// SIMATIC STEP 7 (V5.x) project PLC_KIP
// CPU: CPU 317-2 PN/DP
// station: Hardware
// station: VIPA
// station: P_ADR_BUS
// program: S7 Program(1)

SYMBOL_TABLE
"empty_C0"	C 0	COUNTER
"dFilt_cnt"	C 1	COUNTER
"COM"	DB 100	DB 100
"znm15_pid"	DB 500	FB 58
"CV_dConc1_pid"	DB 501	FB 58
"zadv_riv_nya"	DB 502	FB 58
"Dat_Filt"	FB 1	FB 1
"MD_to_MW"	FB 2	FB 2
"DO_Control"	FB 3	FB 3
"DI_DO_STATE"	FB 4	FB 4
"PID_AO_control"	FB 5	FB 5
"dat_alm"	FB 6	FB 6
"PUT"	FB 15	FB 15	// Write Data to a Remote CPU
"TCONT_CP"	FB 58	FB 58	// temperature PID controller with pulse generator and self-tuning
"DO_MANUAL"	FC 1	FC 1
"SCALE"	FC 105	FC 105	// Scaling Values
"UNSCALE"	FC 106	FC 106	// Unscaling Values
"btn_kvit"	M 3998.0	BOOL
"ZNM15_HM"	M 6000.1	BOOL
"CYCL_EXC"	OB 1	OB 1	// Cycle Execution
"CYC_INT5"	OB 35	OB 35	// Cyclic Interrupt 5
"AIt1_1"	PIW 272	INT
"AIt1_2"	PIW 274	INT
"AIt1_3"	PIW 276	INT
"AIt1_4"	PIW 278	INT
"AIt2_1"	PIW 280	INT
"AIt2_2"	PIW 282	INT
"AIt2_3"	PIW 284	INT
"AIt2_4"	PIW 286	INT
"AIt_3_1"	PIW 288	INT
"AIt_3_2"	PIW 290	INT
"AIt3_3"	PIW 292	INT
"AIt3_4"	PIW 294	INT
"ZN1_cur"	PIW 304	INT
"UVK2_cur"	PIW 306	INT
"UVK1_cur"	PIW 308	INT
"UZ1_in"	PIW 310	INT
"UZ1_out"	PIW 312	INT
"vak_suk1"	PIW 314	INT
"Pidsit_riv"	PIW 316	INT
"vak_suk2"	PIW 318	INT
"vak_suk3"	PIW 320	INT
"vak_suk5"	PIW 322	INT
"vak_suk4"	PIW 324	INT
"vak_suk6"	PIW 326	INT
"vak_val1"	PIW 328	INT
"vak_VN5"	PIW 330	INT
"vak_val2"	PIW 332	INT
"BM8_riv"	PIW 334	INT
"BO9_riv"	PIW 336	INT
"BB11_riv"	PIW 338	INT
"BZ10_riv"	PIW 340	INT
"Gauch_riv"	PIW 342	INT
"NC32"	PIW 344	INT
"Priam_riv"	PIW 346	INT
"NC35"	PIW 348	INT
"GRG_riv"	PIW 350	INT
"vak_VN1"	PIW 352	INT
"vak_VN3"	PIW 354	INT
"vak_VN2"	PIW 356	INT
"vak_VN4"	PIW 358	INT
"dUVK1_in"	PIW 376	INT
"dUVK2_in"	PIW 378	INT
"dC8_in"	PIW 380	INT
"dUVK1_out"	PIW 382	INT
"dUVK2_out"	PIW 384	INT
"dC8_out"	PIW 386	INT
"dSUM_pr"	PIW 388	INT
"AI2_4"	PIW 390	INT
"dRivSkop"	PIW 392	INT
"dRIV_NYA"	PIW 394	INT
"dRivPidNya"	PIW 396	INT
"dUzloulov_in"	PIW 398	INT
"dMlyn_in"	PIW 400	INT
"AI4_2"	PIW 402	INT
"dMlyn_out"	PIW 404	INT
"dUzloulov_out"	PIW 406	INT
"taskZNM12"	PQW 272	INT
"ZasNV23_1"	PQW 274	INT
"taskZNM15"	PQW 276	INT
"reg_knctr2"	PQW 278	INT
"zadv_recycl_nya"	PQW 296	INT
"CV_conc1"	PQW 300	INT
"GET"	SFB 14	SFB 14	// Read Data From a Remote CPU
"empty_T0"	T 0	TIMER
"dFilt_tmr"	T 1	TIMER
"VAT_3_kip"	VAT 1	
"VAT_4"	VAT 2	
"VAT_3_HI_LOW_Dat"	VAT 3	
END_SYMBOL_TABLE

FUNCTION_BLOCK "Dat_Filt"	// FB 1
TITLE = Чтение датчика
//**********************************
VERSION : 0.1
VAR_INPUT
  dPIW : INT ;
  dHi_lim : DINT ;
  dLow_lim : DINT ;
  dErr_lvl : INT ;
  Sample : S5TIME ;
END_VAR
VAR_OUTPUT
  Dat_err : BOOL ;
  Dat_f : REAL ;
  Dat_md : DINT ;
END_VAR
VAR
  Bipolar : BOOL ;
  rst_T1 : BOOL ;
  int_C1 : INT ;
  Hi_lim_re : REAL ;
  Low_lim_re : REAL ;
  DAT_re : REAL ;
  DAT_avg : REAL ;
  dat_re0 : REAL ;
  dat_re1 : REAL ;
  dat_re2 : REAL ;
  dat_re3 : REAL ;
  dat_re4 : REAL ;
  dat_re5 : REAL ;
  dat_re6 : REAL ;
  dat_re7 : REAL ;
  dat_re8 : REAL ;
  dat_re9 : REAL ;
  sum : REAL ;
END_VAR
VAR_TEMP
  SCL_err : WORD ;
  UNSCL_err : WORD ;
END_VAR
BEGIN
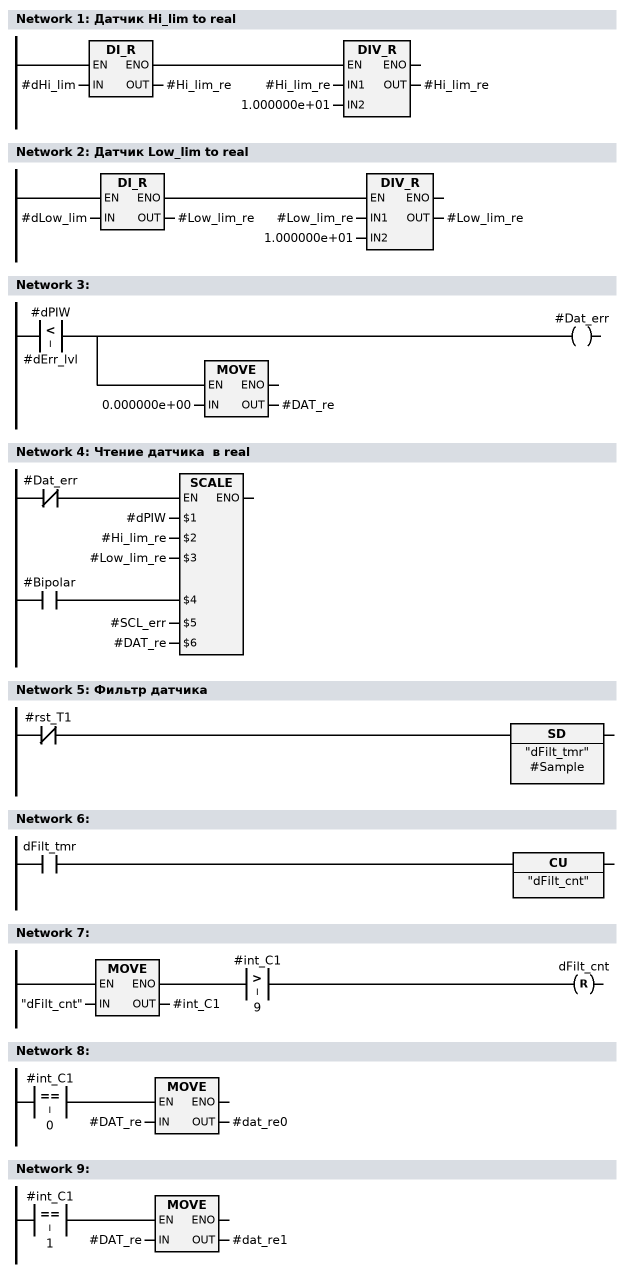
NETWORK
TITLE = Датчик Hi_lim to real
      A(;
      L     #dHi_lim;
      DTR;
      T     #Hi_lim_re;
      SET;
      SAVE;
      CLR;
      A     BR;
      );
      JNB   _001;
      L     #Hi_lim_re;
      L     1.000000e+01;
      /R;
      T     #Hi_lim_re;
_001: NOP   0;
NETWORK
TITLE = Датчик Low_lim to real
      A(;
      L     #dLow_lim;
      DTR;
      T     #Low_lim_re;
      SET;
      SAVE;
      CLR;
      A     BR;
      );
      JNB   _002;
      L     #Low_lim_re;
      L     1.000000e+01;
      /R;
      T     #Low_lim_re;
_002: NOP   0;
NETWORK
TITLE =
//Ошибка чтения датчика
      L     #dPIW;
      L     #dErr_lvl;
      <I;
      =     L 4.0;
      A     L 4.0;
      BLD   102;
      =     #Dat_err;
      A     L 4.0;
      JNB   _003;
      L     0.000000e+00;
      T     #DAT_re;
_003: NOP   0;
NETWORK
TITLE = Чтение датчика  в real
      A     #Bipolar;
      =     L 4.0;
      BLD   103;
      AN    #Dat_err;
      JNB   _004;
      CALL  "SCALE" (
           $1                       := #dPIW,
           $2                       := #Hi_lim_re,
           $3                       := #Low_lim_re,
           $4                       := L 4.0,
           $5                       := #SCL_err,
           $6                       := #DAT_re);
_004: NOP   0;
NETWORK
TITLE = Фильтр датчика
//***************************************************
      AN    #rst_T1;
      L     #Sample;
      SD    "dFilt_tmr";
NETWORK
TITLE =
      A     "dFilt_tmr";
      CU    "dFilt_cnt";
NETWORK
TITLE =
      A(;
      L     "dFilt_cnt";
      T     #int_C1;
      SET;
      SAVE;
      CLR;
      A     BR;
      );
      A(;
      L     #int_C1;
      L     9;
      >I;
      );
      R     "dFilt_cnt";
NETWORK
TITLE =
      A(;
      L     #int_C1;
      L     0;
      ==I;
      );
      JNB   _005;
      L     #DAT_re;
      T     #dat_re0;
_005: NOP   0;
NETWORK
TITLE =
      A(;
      L     #int_C1;
      L     1;
      ==I;
      );
      JNB   _006;
      L     #DAT_re;
      T     #dat_re1;
_006: NOP   0;
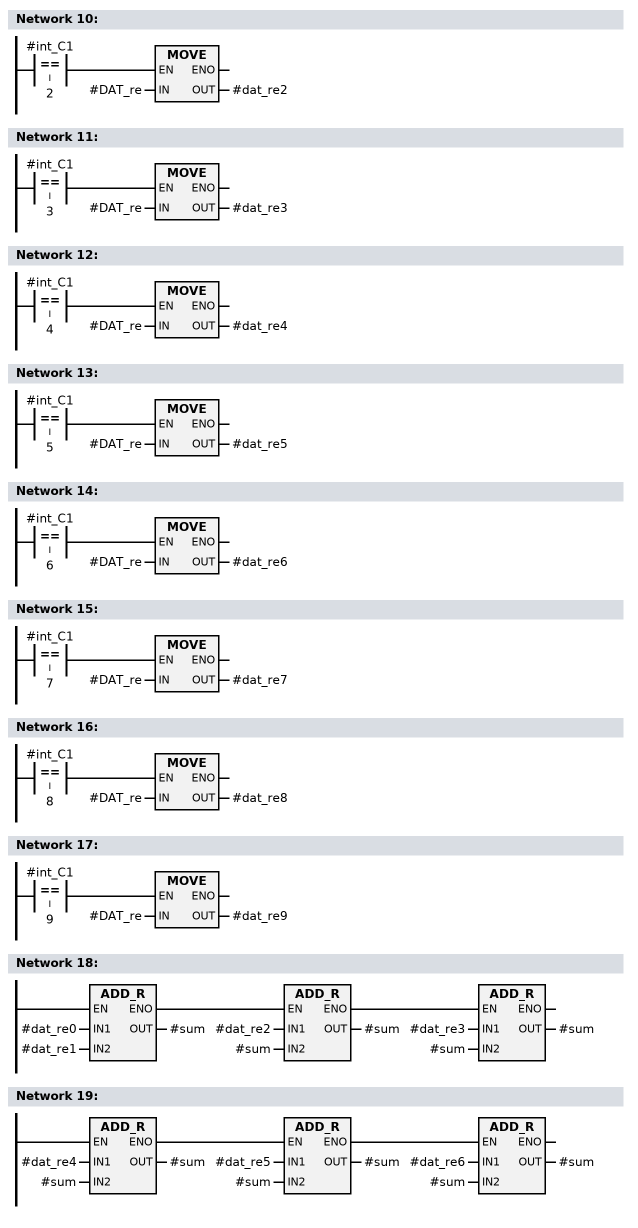
NETWORK
TITLE =
      A(;
      L     #int_C1;
      L     2;
      ==I;
      );
      JNB   _007;
      L     #DAT_re;
      T     #dat_re2;
_007: NOP   0;
NETWORK
TITLE =
      A(;
      L     #int_C1;
      L     3;
      ==I;
      );
      JNB   _008;
      L     #DAT_re;
      T     #dat_re3;
_008: NOP   0;
NETWORK
TITLE =
      A(;
      L     #int_C1;
      L     4;
      ==I;
      );
      JNB   _009;
      L     #DAT_re;
      T     #dat_re4;
_009: NOP   0;
NETWORK
TITLE =
      A(;
      L     #int_C1;
      L     5;
      ==I;
      );
      JNB   _00a;
      L     #DAT_re;
      T     #dat_re5;
_00a: NOP   0;
NETWORK
TITLE =
      A(;
      L     #int_C1;
      L     6;
      ==I;
      );
      JNB   _00b;
      L     #DAT_re;
      T     #dat_re6;
_00b: NOP   0;
NETWORK
TITLE =
      A(;
      L     #int_C1;
      L     7;
      ==I;
      );
      JNB   _00c;
      L     #DAT_re;
      T     #dat_re7;
_00c: NOP   0;
NETWORK
TITLE =
      A(;
      L     #int_C1;
      L     8;
      ==I;
      );
      JNB   _00d;
      L     #DAT_re;
      T     #dat_re8;
_00d: NOP   0;
NETWORK
TITLE =
      A(;
      L     #int_C1;
      L     9;
      ==I;
      );
      JNB   _00e;
      L     #DAT_re;
      T     #dat_re9;
_00e: NOP   0;
NETWORK
TITLE =
      A(;
      A(;
      L     #dat_re0;
      L     #dat_re1;
      +R;
      T     #sum;
      AN    OV;
      SAVE;
      CLR;
      A     BR;
      );
      JNB   _00f;
      L     #dat_re2;
      L     #sum;
      +R;
      T     #sum;
      AN    OV;
      SAVE;
      CLR;
_00f: A     BR;
      );
      JNB   _010;
      L     #dat_re3;
      L     #sum;
      +R;
      T     #sum;
_010: NOP   0;
NETWORK
TITLE =
      A(;
      A(;
      L     #dat_re4;
      L     #sum;
      +R;
      T     #sum;
      AN    OV;
      SAVE;
      CLR;
      A     BR;
      );
      JNB   _011;
      L     #dat_re5;
      L     #sum;
      +R;
      T     #sum;
      AN    OV;
      SAVE;
      CLR;
_011: A     BR;
      );
      JNB   _012;
      L     #dat_re6;
      L     #sum;
      +R;
      T     #sum;
_012: NOP   0;
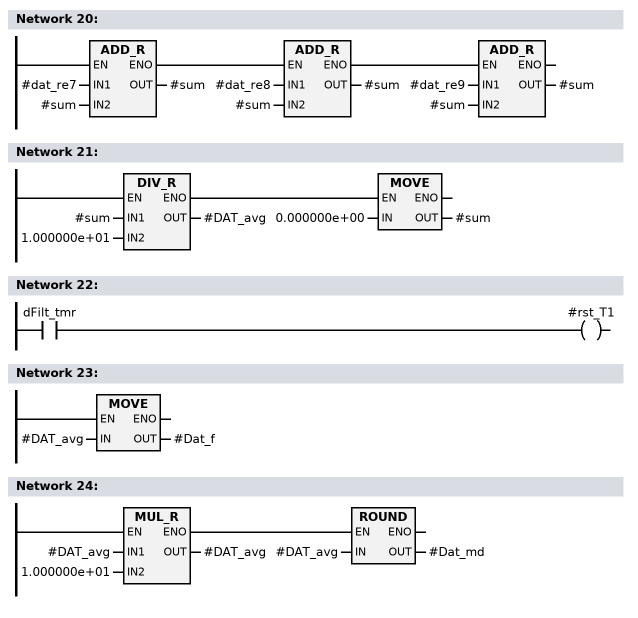
NETWORK
TITLE =
      A(;
      A(;
      L     #dat_re7;
      L     #sum;
      +R;
      T     #sum;
      AN    OV;
      SAVE;
      CLR;
      A     BR;
      );
      JNB   _013;
      L     #dat_re8;
      L     #sum;
      +R;
      T     #sum;
      AN    OV;
      SAVE;
      CLR;
_013: A     BR;
      );
      JNB   _014;
      L     #dat_re9;
      L     #sum;
      +R;
      T     #sum;
_014: NOP   0;
NETWORK
TITLE =
      A(;
      L     #sum;
      L     1.000000e+01;
      /R;
      T     #DAT_avg;
      AN    OV;
      SAVE;
      CLR;
      A     BR;
      );
      JNB   _015;
      L     0.000000e+00;
      T     #sum;
_015: NOP   0;
NETWORK
TITLE =
      A     "dFilt_tmr";
      =     #rst_T1;
NETWORK
TITLE =
      L     #DAT_avg;
      T     #Dat_f;
      NOP   0;
NETWORK
TITLE =
      A(;
      L     #DAT_avg;
      L     1.000000e+01;
      *R;
      T     #DAT_avg;
      AN    OV;
      SAVE;
      CLR;
      A     BR;
      );
      JNB   _016;
      L     #DAT_avg;
      RND;
      T     #Dat_md;
_016: NOP   0;
END_FUNCTION_BLOCK

FUNCTION_BLOCK "MD_to_MW"	// FB 2
//Для обміну між ПЛК КІП та ПЛК ДВГ (з MD в MW)
VERSION : 0.1
VAR_TEMP
  ZNM15_task_re : REAL ;
  cv_conc1_task_re : REAL ;
  cv_recycle_task_re : REAL ;
END_VAR
BEGIN
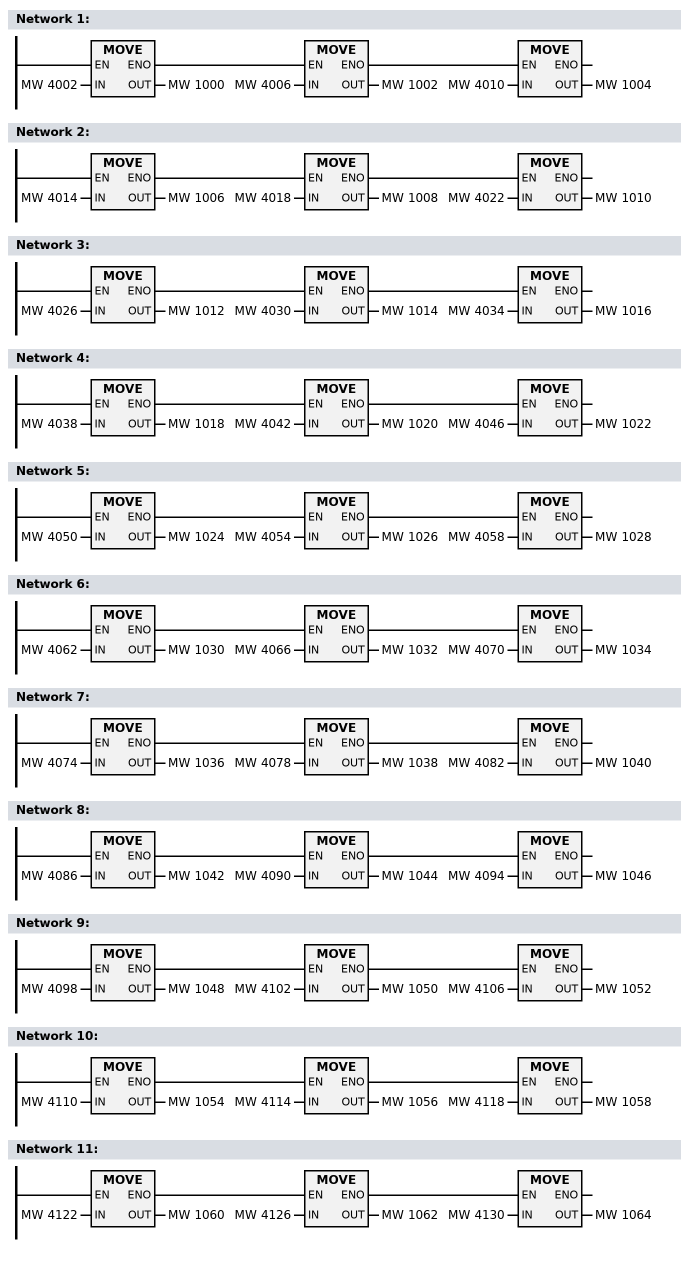
NETWORK
TITLE =
      A(;
      A(;
      L     MW 4002;
      T     MW 1000;
      SET;
      SAVE;
      CLR;
      A     BR;
      );
      JNB   _001;
      L     MW 4006;
      T     MW 1002;
      SET;
      SAVE;
      CLR;
_001: A     BR;
      );
      JNB   _002;
      L     MW 4010;
      T     MW 1004;
_002: NOP   0;
NETWORK
TITLE =
      A(;
      A(;
      L     MW 4014;
      T     MW 1006;
      SET;
      SAVE;
      CLR;
      A     BR;
      );
      JNB   _003;
      L     MW 4018;
      T     MW 1008;
      SET;
      SAVE;
      CLR;
_003: A     BR;
      );
      JNB   _004;
      L     MW 4022;
      T     MW 1010;
_004: NOP   0;
NETWORK
TITLE =
      A(;
      A(;
      L     MW 4026;
      T     MW 1012;
      SET;
      SAVE;
      CLR;
      A     BR;
      );
      JNB   _005;
      L     MW 4030;
      T     MW 1014;
      SET;
      SAVE;
      CLR;
_005: A     BR;
      );
      JNB   _006;
      L     MW 4034;
      T     MW 1016;
_006: NOP   0;
NETWORK
TITLE =
      A(;
      A(;
      L     MW 4038;
      T     MW 1018;
      SET;
      SAVE;
      CLR;
      A     BR;
      );
      JNB   _007;
      L     MW 4042;
      T     MW 1020;
      SET;
      SAVE;
      CLR;
_007: A     BR;
      );
      JNB   _008;
      L     MW 4046;
      T     MW 1022;
_008: NOP   0;
NETWORK
TITLE =
      A(;
      A(;
      L     MW 4050;
      T     MW 1024;
      SET;
      SAVE;
      CLR;
      A     BR;
      );
      JNB   _009;
      L     MW 4054;
      T     MW 1026;
      SET;
      SAVE;
      CLR;
_009: A     BR;
      );
      JNB   _00a;
      L     MW 4058;
      T     MW 1028;
_00a: NOP   0;
NETWORK
TITLE =
      A(;
      A(;
      L     MW 4062;
      T     MW 1030;
      SET;
      SAVE;
      CLR;
      A     BR;
      );
      JNB   _00b;
      L     MW 4066;
      T     MW 1032;
      SET;
      SAVE;
      CLR;
_00b: A     BR;
      );
      JNB   _00c;
      L     MW 4070;
      T     MW 1034;
_00c: NOP   0;
NETWORK
TITLE =
      A(;
      A(;
      L     MW 4074;
      T     MW 1036;
      SET;
      SAVE;
      CLR;
      A     BR;
      );
      JNB   _00d;
      L     MW 4078;
      T     MW 1038;
      SET;
      SAVE;
      CLR;
_00d: A     BR;
      );
      JNB   _00e;
      L     MW 4082;
      T     MW 1040;
_00e: NOP   0;
NETWORK
TITLE =
      A(;
      A(;
      L     MW 4086;
      T     MW 1042;
      SET;
      SAVE;
      CLR;
      A     BR;
      );
      JNB   _00f;
      L     MW 4090;
      T     MW 1044;
      SET;
      SAVE;
      CLR;
_00f: A     BR;
      );
      JNB   _010;
      L     MW 4094;
      T     MW 1046;
_010: NOP   0;
NETWORK
TITLE =
      A(;
      A(;
      L     MW 4098;
      T     MW 1048;
      SET;
      SAVE;
      CLR;
      A     BR;
      );
      JNB   _011;
      L     MW 4102;
      T     MW 1050;
      SET;
      SAVE;
      CLR;
_011: A     BR;
      );
      JNB   _012;
      L     MW 4106;
      T     MW 1052;
_012: NOP   0;
NETWORK
TITLE =
      A(;
      A(;
      L     MW 4110;
      T     MW 1054;
      SET;
      SAVE;
      CLR;
      A     BR;
      );
      JNB   _013;
      L     MW 4114;
      T     MW 1056;
      SET;
      SAVE;
      CLR;
_013: A     BR;
      );
      JNB   _014;
      L     MW 4118;
      T     MW 1058;
_014: NOP   0;
NETWORK
TITLE =
      A(;
      A(;
      L     MW 4122;
      T     MW 1060;
      SET;
      SAVE;
      CLR;
      A     BR;
      );
      JNB   _015;
      L     MW 4126;
      T     MW 1062;
      SET;
      SAVE;
      CLR;
_015: A     BR;
      );
      JNB   _016;
      L     MW 4130;
      T     MW 1064;
_016: NOP   0;
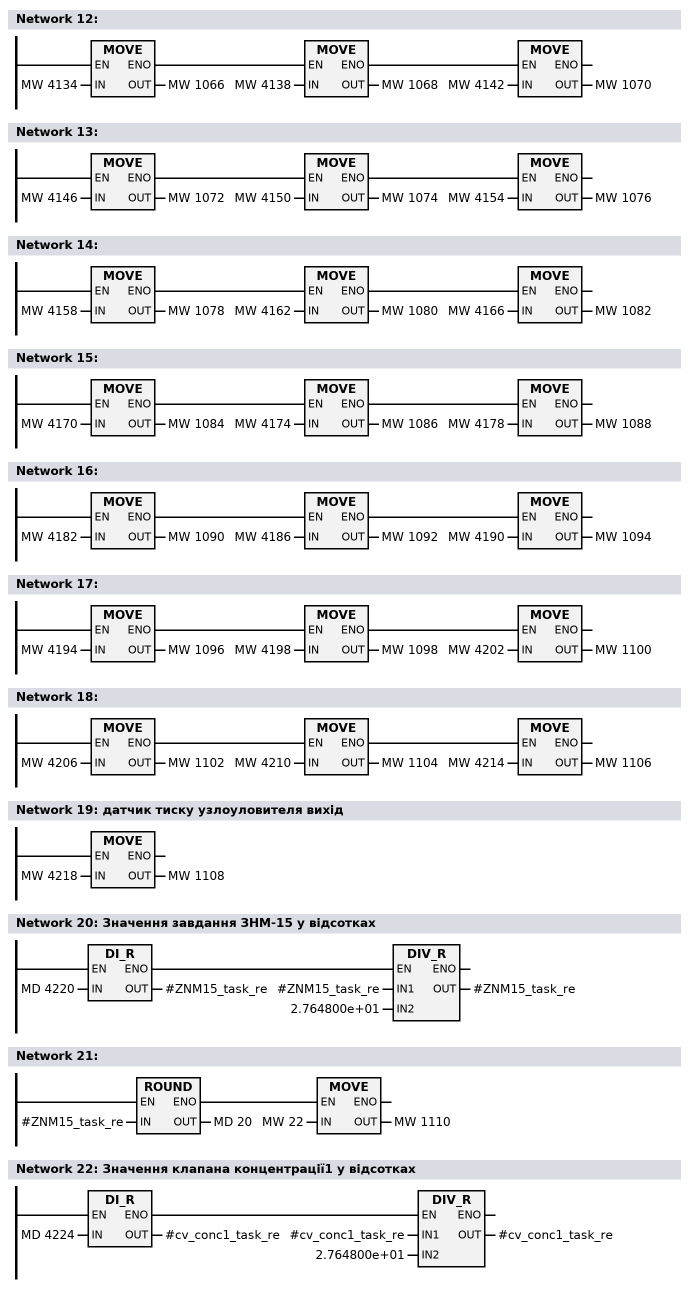
NETWORK
TITLE =
      A(;
      A(;
      L     MW 4134;
      T     MW 1066;
      SET;
      SAVE;
      CLR;
      A     BR;
      );
      JNB   _017;
      L     MW 4138;
      T     MW 1068;
      SET;
      SAVE;
      CLR;
_017: A     BR;
      );
      JNB   _018;
      L     MW 4142;
      T     MW 1070;
_018: NOP   0;
NETWORK
TITLE =
      A(;
      A(;
      L     MW 4146;
      T     MW 1072;
      SET;
      SAVE;
      CLR;
      A     BR;
      );
      JNB   _019;
      L     MW 4150;
      T     MW 1074;
      SET;
      SAVE;
      CLR;
_019: A     BR;
      );
      JNB   _01a;
      L     MW 4154;
      T     MW 1076;
_01a: NOP   0;
NETWORK
TITLE =
      A(;
      A(;
      L     MW 4158;
      T     MW 1078;
      SET;
      SAVE;
      CLR;
      A     BR;
      );
      JNB   _01b;
      L     MW 4162;
      T     MW 1080;
      SET;
      SAVE;
      CLR;
_01b: A     BR;
      );
      JNB   _01c;
      L     MW 4166;
      T     MW 1082;
_01c: NOP   0;
NETWORK
TITLE =
      A(;
      A(;
      L     MW 4170;
      T     MW 1084;
      SET;
      SAVE;
      CLR;
      A     BR;
      );
      JNB   _01d;
      L     MW 4174;
      T     MW 1086;
      SET;
      SAVE;
      CLR;
_01d: A     BR;
      );
      JNB   _01e;
      L     MW 4178;
      T     MW 1088;
_01e: NOP   0;
NETWORK
TITLE =
      A(;
      A(;
      L     MW 4182;
      T     MW 1090;
      SET;
      SAVE;
      CLR;
      A     BR;
      );
      JNB   _01f;
      L     MW 4186;
      T     MW 1092;
      SET;
      SAVE;
      CLR;
_01f: A     BR;
      );
      JNB   _020;
      L     MW 4190;
      T     MW 1094;
_020: NOP   0;
NETWORK
TITLE =
      A(;
      A(;
      L     MW 4194;
      T     MW 1096;
      SET;
      SAVE;
      CLR;
      A     BR;
      );
      JNB   _021;
      L     MW 4198;
      T     MW 1098;
      SET;
      SAVE;
      CLR;
_021: A     BR;
      );
      JNB   _022;
      L     MW 4202;
      T     MW 1100;
_022: NOP   0;
NETWORK
TITLE =
      A(;
      A(;
      L     MW 4206;
      T     MW 1102;
      SET;
      SAVE;
      CLR;
      A     BR;
      );
      JNB   _023;
      L     MW 4210;
      T     MW 1104;
      SET;
      SAVE;
      CLR;
_023: A     BR;
      );
      JNB   _024;
      L     MW 4214;
      T     MW 1106;
_024: NOP   0;
NETWORK
TITLE = датчик тиску узлоуловителя вихід
      L     MW 4218;
      T     MW 1108;
      NOP   0;
NETWORK
TITLE = Значення завдання ЗНМ-15 у відсотках
//Значення завдання ЗНМ-15 у відсотках
      A(;
      L     MD 4220;
      DTR;
      T     #ZNM15_task_re;
      SET;
      SAVE;
      CLR;
      A     BR;
      );
      JNB   _025;
      L     #ZNM15_task_re;
      L     2.764800e+01;
      /R;
      T     #ZNM15_task_re;
_025: NOP   0;
NETWORK
TITLE =
      A(;
      L     #ZNM15_task_re;
      RND;
      T     MD 20;
      AN    OV;
      SAVE;
      CLR;
      A     BR;
      );
      JNB   _026;
      L     MW 22;
      T     MW 1110;
_026: NOP   0;
NETWORK
TITLE = Значення клапана концентрації1 у відсотках
      A(;
      L     MD 4224;
      DTR;
      T     #cv_conc1_task_re;
      SET;
      SAVE;
      CLR;
      A     BR;
      );
      JNB   _027;
      L     #cv_conc1_task_re;
      L     2.764800e+01;
      /R;
      T     #cv_conc1_task_re;
_027: NOP   0;
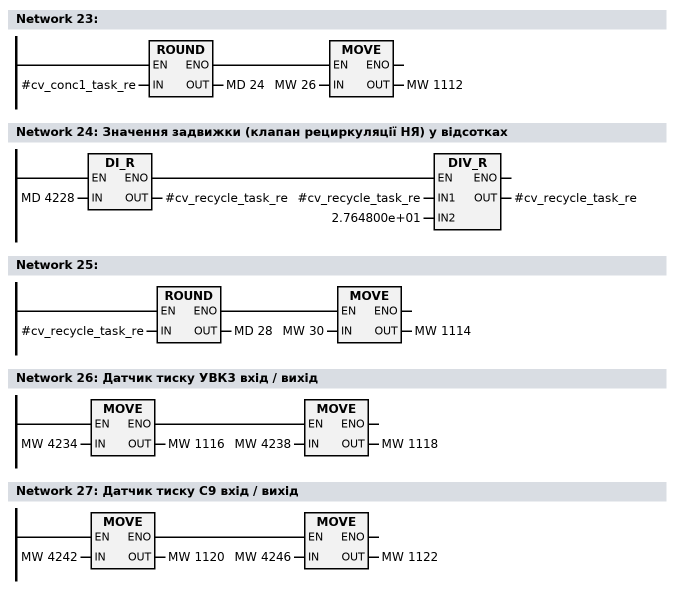
NETWORK
TITLE =
      A(;
      L     #cv_conc1_task_re;
      RND;
      T     MD 24;
      AN    OV;
      SAVE;
      CLR;
      A     BR;
      );
      JNB   _028;
      L     MW 26;
      T     MW 1112;
_028: NOP   0;
NETWORK
TITLE = Значення задвижки (клапан рециркуляції НЯ) у відсотках
      A(;
      L     MD 4228;
      DTR;
      T     #cv_recycle_task_re;
      SET;
      SAVE;
      CLR;
      A     BR;
      );
      JNB   _029;
      L     #cv_recycle_task_re;
      L     2.764800e+01;
      /R;
      T     #cv_recycle_task_re;
_029: NOP   0;
NETWORK
TITLE =
      A(;
      L     #cv_recycle_task_re;
      RND;
      T     MD 28;
      AN    OV;
      SAVE;
      CLR;
      A     BR;
      );
      JNB   _02a;
      L     MW 30;
      T     MW 1114;
_02a: NOP   0;
NETWORK
TITLE = Датчик тиску УВК3 вхід / вихід
      A(;
      L     MW 4234;
      T     MW 1116;
      SET;
      SAVE;
      CLR;
      A     BR;
      );
      JNB   _02b;
      L     MW 4238;
      T     MW 1118;
_02b: NOP   0;
NETWORK
TITLE = Датчик тиску C9 вхід / вихід
      A(;
      L     MW 4242;
      T     MW 1120;
      SET;
      SAVE;
      CLR;
      A     BR;
      );
      JNB   _02c;
      L     MW 4246;
      T     MW 1122;
_02c: NOP   0;
END_FUNCTION_BLOCK

FUNCTION_BLOCK "DO_Control"	// FB 3
//Керування дискретними виходами
VERSION : 0.1
BEGIN
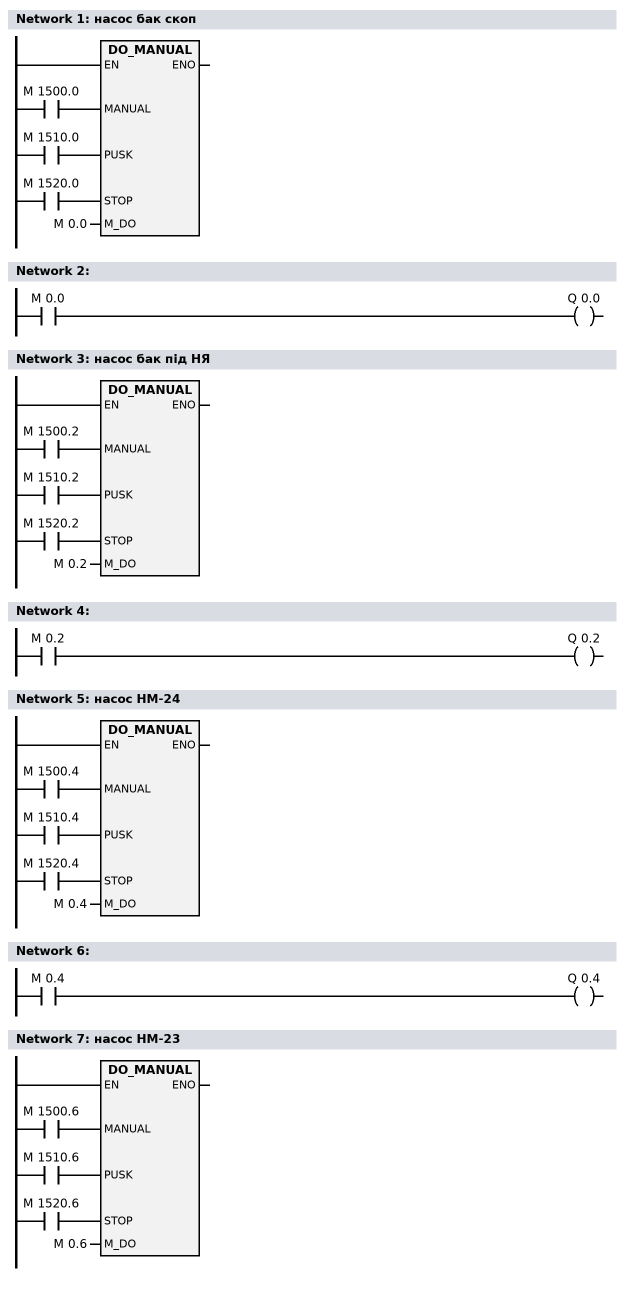
NETWORK
TITLE = насос бак скоп
      A     M 1500.0;
      =     L 0.0;
      BLD   103;
      A     M 1510.0;
      =     L 0.1;
      BLD   103;
      A     M 1520.0;
      =     L 0.2;
      BLD   103;
      CALL  "DO_MANUAL" (
           MANUAL                   := L 0.0,
           PUSK                     := L 0.1,
           STOP                     := L 0.2,
           M_DO                     := M 0.0);
      NOP   0;
NETWORK
TITLE =
      A     M 0.0;
      =     Q 0.0;
NETWORK
TITLE = насос бак під НЯ
      A     M 1500.2;
      =     L 0.0;
      BLD   103;
      A     M 1510.2;
      =     L 0.1;
      BLD   103;
      A     M 1520.2;
      =     L 0.2;
      BLD   103;
      CALL  "DO_MANUAL" (
           MANUAL                   := L 0.0,
           PUSK                     := L 0.1,
           STOP                     := L 0.2,
           M_DO                     := M 0.2);
      NOP   0;
NETWORK
TITLE =
      A     M 0.2;
      =     Q 0.2;
NETWORK
TITLE = насос НМ-24
      A     M 1500.4;
      =     L 0.0;
      BLD   103;
      A     M 1510.4;
      =     L 0.1;
      BLD   103;
      A     M 1520.4;
      =     L 0.2;
      BLD   103;
      CALL  "DO_MANUAL" (
           MANUAL                   := L 0.0,
           PUSK                     := L 0.1,
           STOP                     := L 0.2,
           M_DO                     := M 0.4);
      NOP   0;
NETWORK
TITLE =
      A     M 0.4;
      =     Q 0.4;
NETWORK
TITLE = насос НМ-23
      A     M 1500.6;
      =     L 0.0;
      BLD   103;
      A     M 1510.6;
      =     L 0.1;
      BLD   103;
      A     M 1520.6;
      =     L 0.2;
      BLD   103;
      CALL  "DO_MANUAL" (
           MANUAL                   := L 0.0,
           PUSK                     := L 0.1,
           STOP                     := L 0.2,
           M_DO                     := M 0.6);
      NOP   0;
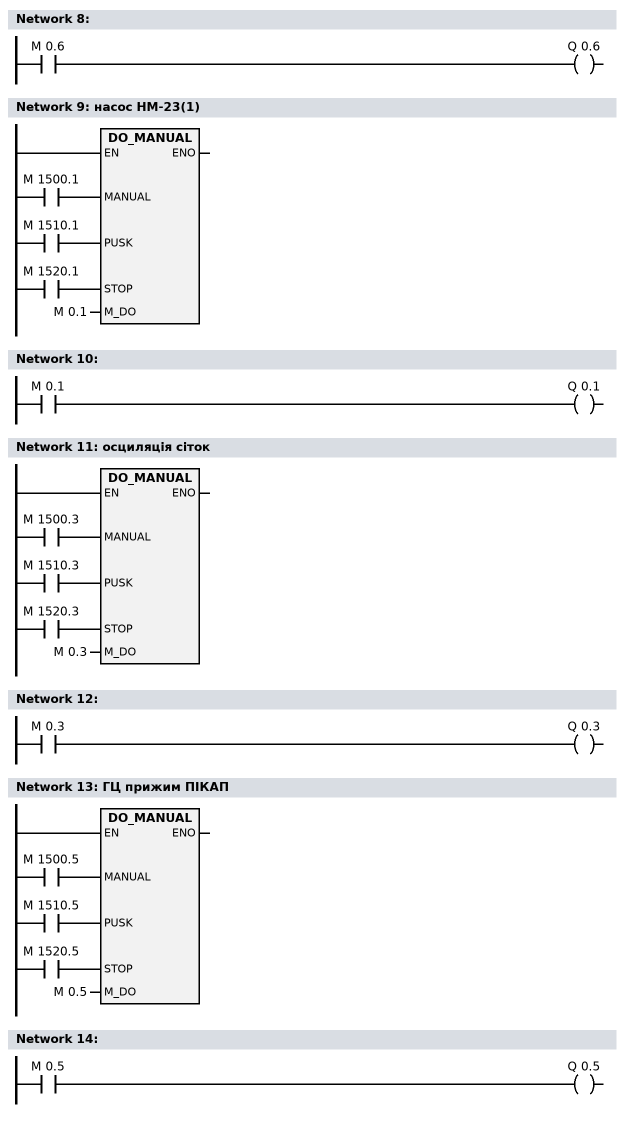
NETWORK
TITLE =
      A     M 0.6;
      =     Q 0.6;
NETWORK
TITLE = насос НМ-23(1)
      A     M 1500.1;
      =     L 0.0;
      BLD   103;
      A     M 1510.1;
      =     L 0.1;
      BLD   103;
      A     M 1520.1;
      =     L 0.2;
      BLD   103;
      CALL  "DO_MANUAL" (
           MANUAL                   := L 0.0,
           PUSK                     := L 0.1,
           STOP                     := L 0.2,
           M_DO                     := M 0.1);
      NOP   0;
NETWORK
TITLE =
      A     M 0.1;
      =     Q 0.1;
NETWORK
TITLE = осциляція сіток
      A     M 1500.3;
      =     L 0.0;
      BLD   103;
      A     M 1510.3;
      =     L 0.1;
      BLD   103;
      A     M 1520.3;
      =     L 0.2;
      BLD   103;
      CALL  "DO_MANUAL" (
           MANUAL                   := L 0.0,
           PUSK                     := L 0.1,
           STOP                     := L 0.2,
           M_DO                     := M 0.3);
      NOP   0;
NETWORK
TITLE =
      A     M 0.3;
      =     Q 0.3;
NETWORK
TITLE = ГЦ прижим ПІКАП
      A     M 1500.5;
      =     L 0.0;
      BLD   103;
      A     M 1510.5;
      =     L 0.1;
      BLD   103;
      A     M 1520.5;
      =     L 0.2;
      BLD   103;
      CALL  "DO_MANUAL" (
           MANUAL                   := L 0.0,
           PUSK                     := L 0.1,
           STOP                     := L 0.2,
           M_DO                     := M 0.5);
      NOP   0;
NETWORK
TITLE =
      A     M 0.5;
      =     Q 0.5;
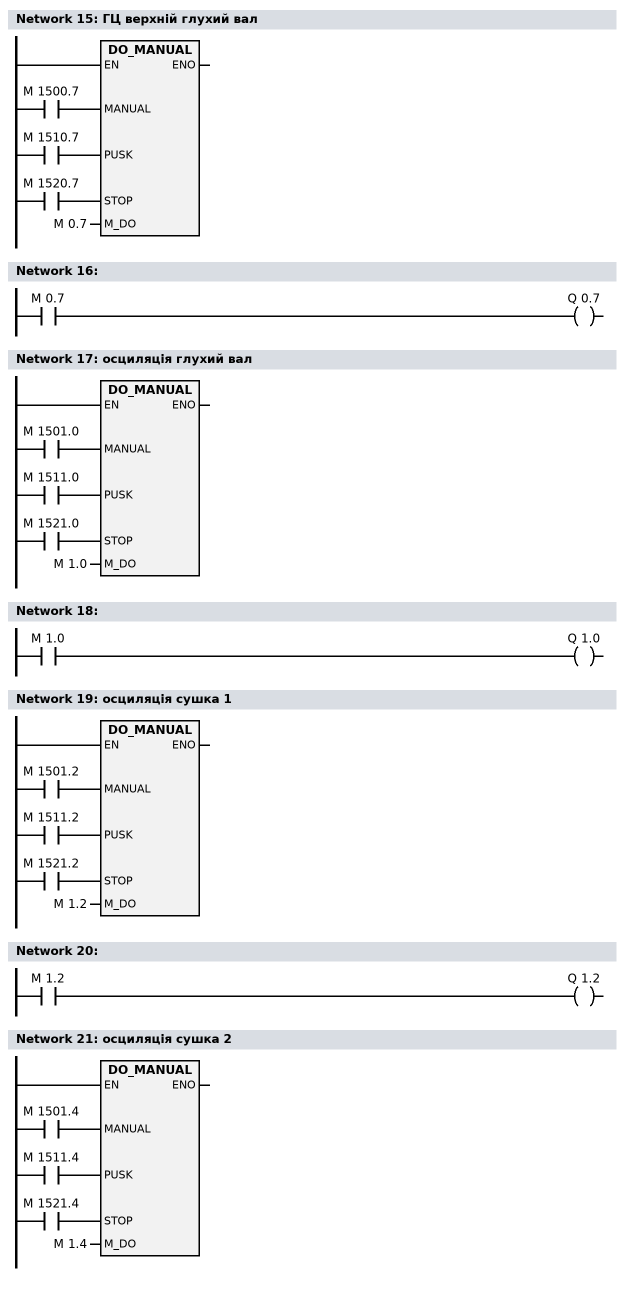
NETWORK
TITLE = ГЦ верхній глухий вал
      A     M 1500.7;
      =     L 0.0;
      BLD   103;
      A     M 1510.7;
      =     L 0.1;
      BLD   103;
      A     M 1520.7;
      =     L 0.2;
      BLD   103;
      CALL  "DO_MANUAL" (
           MANUAL                   := L 0.0,
           PUSK                     := L 0.1,
           STOP                     := L 0.2,
           M_DO                     := M 0.7);
      NOP   0;
NETWORK
TITLE =
      A     M 0.7;
      =     Q 0.7;
NETWORK
TITLE = осциляція глухий вал
      A     M 1501.0;
      =     L 0.0;
      BLD   103;
      A     M 1511.0;
      =     L 0.1;
      BLD   103;
      A     M 1521.0;
      =     L 0.2;
      BLD   103;
      CALL  "DO_MANUAL" (
           MANUAL                   := L 0.0,
           PUSK                     := L 0.1,
           STOP                     := L 0.2,
           M_DO                     := M 1.0);
      NOP   0;
NETWORK
TITLE =
      A     M 1.0;
      =     Q 1.0;
NETWORK
TITLE = осциляція сушка 1
      A     M 1501.2;
      =     L 0.0;
      BLD   103;
      A     M 1511.2;
      =     L 0.1;
      BLD   103;
      A     M 1521.2;
      =     L 0.2;
      BLD   103;
      CALL  "DO_MANUAL" (
           MANUAL                   := L 0.0,
           PUSK                     := L 0.1,
           STOP                     := L 0.2,
           M_DO                     := M 1.2);
      NOP   0;
NETWORK
TITLE =
      A     M 1.2;
      =     Q 1.2;
NETWORK
TITLE = осциляція сушка 2
      A     M 1501.4;
      =     L 0.0;
      BLD   103;
      A     M 1511.4;
      =     L 0.1;
      BLD   103;
      A     M 1521.4;
      =     L 0.2;
      BLD   103;
      CALL  "DO_MANUAL" (
           MANUAL                   := L 0.0,
           PUSK                     := L 0.1,
           STOP                     := L 0.2,
           M_DO                     := M 1.4);
      NOP   0;
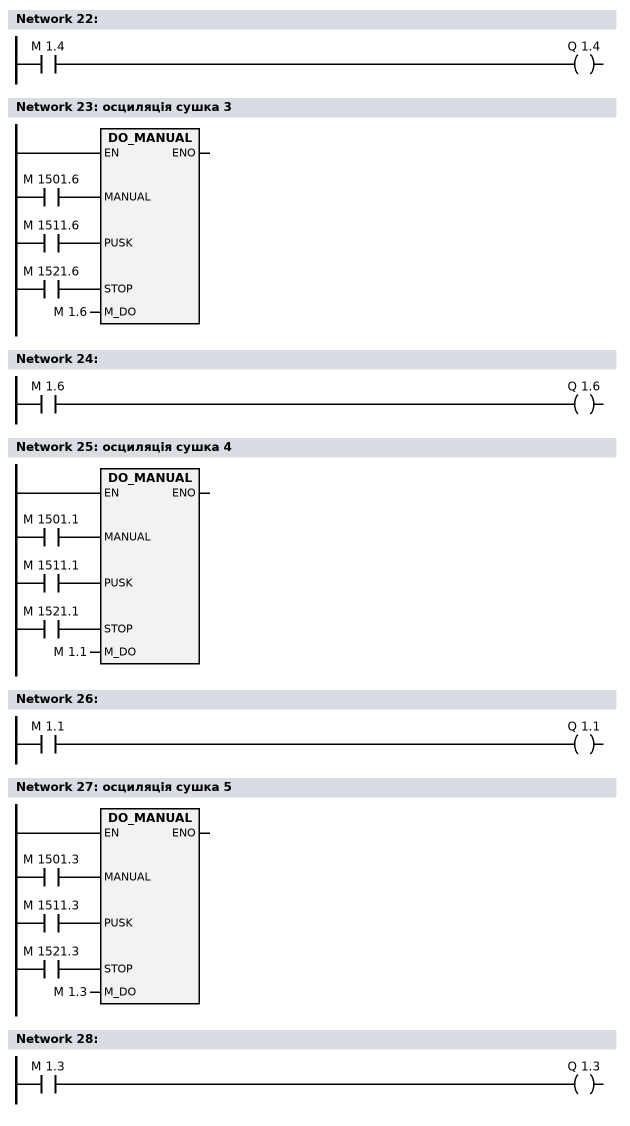
NETWORK
TITLE =
      A     M 1.4;
      =     Q 1.4;
NETWORK
TITLE = осциляція сушка 3
      A     M 1501.6;
      =     L 0.0;
      BLD   103;
      A     M 1511.6;
      =     L 0.1;
      BLD   103;
      A     M 1521.6;
      =     L 0.2;
      BLD   103;
      CALL  "DO_MANUAL" (
           MANUAL                   := L 0.0,
           PUSK                     := L 0.1,
           STOP                     := L 0.2,
           M_DO                     := M 1.6);
      NOP   0;
NETWORK
TITLE =
      A     M 1.6;
      =     Q 1.6;
NETWORK
TITLE = осциляція сушка 4
      A     M 1501.1;
      =     L 0.0;
      BLD   103;
      A     M 1511.1;
      =     L 0.1;
      BLD   103;
      A     M 1521.1;
      =     L 0.2;
      BLD   103;
      CALL  "DO_MANUAL" (
           MANUAL                   := L 0.0,
           PUSK                     := L 0.1,
           STOP                     := L 0.2,
           M_DO                     := M 1.1);
      NOP   0;
NETWORK
TITLE =
      A     M 1.1;
      =     Q 1.1;
NETWORK
TITLE = осциляція сушка 5
      A     M 1501.3;
      =     L 0.0;
      BLD   103;
      A     M 1511.3;
      =     L 0.1;
      BLD   103;
      A     M 1521.3;
      =     L 0.2;
      BLD   103;
      CALL  "DO_MANUAL" (
           MANUAL                   := L 0.0,
           PUSK                     := L 0.1,
           STOP                     := L 0.2,
           M_DO                     := M 1.3);
      NOP   0;
NETWORK
TITLE =
      A     M 1.3;
      =     Q 1.3;
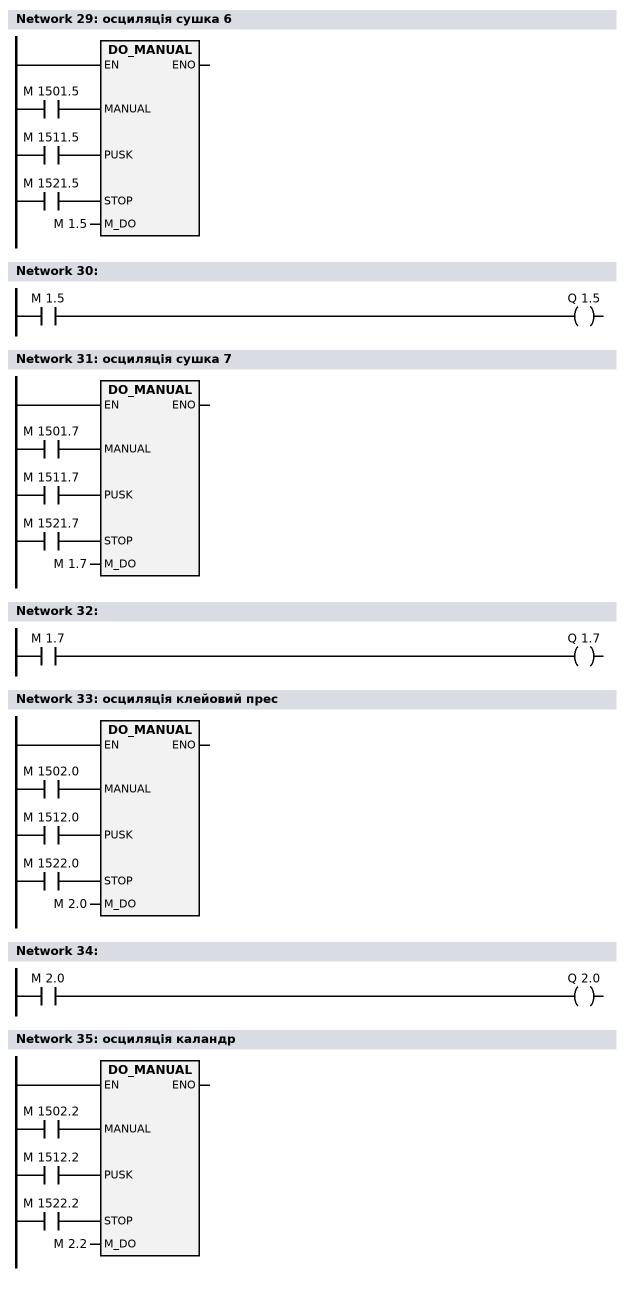
NETWORK
TITLE = осциляція сушка 6
      A     M 1501.5;
      =     L 0.0;
      BLD   103;
      A     M 1511.5;
      =     L 0.1;
      BLD   103;
      A     M 1521.5;
      =     L 0.2;
      BLD   103;
      CALL  "DO_MANUAL" (
           MANUAL                   := L 0.0,
           PUSK                     := L 0.1,
           STOP                     := L 0.2,
           M_DO                     := M 1.5);
      NOP   0;
NETWORK
TITLE =
      A     M 1.5;
      =     Q 1.5;
NETWORK
TITLE = осциляція сушка 7
      A     M 1501.7;
      =     L 0.0;
      BLD   103;
      A     M 1511.7;
      =     L 0.1;
      BLD   103;
      A     M 1521.7;
      =     L 0.2;
      BLD   103;
      CALL  "DO_MANUAL" (
           MANUAL                   := L 0.0,
           PUSK                     := L 0.1,
           STOP                     := L 0.2,
           M_DO                     := M 1.7);
      NOP   0;
NETWORK
TITLE =
      A     M 1.7;
      =     Q 1.7;
NETWORK
TITLE = осциляція клейовий прес
      A     M 1502.0;
      =     L 0.0;
      BLD   103;
      A     M 1512.0;
      =     L 0.1;
      BLD   103;
      A     M 1522.0;
      =     L 0.2;
      BLD   103;
      CALL  "DO_MANUAL" (
           MANUAL                   := L 0.0,
           PUSK                     := L 0.1,
           STOP                     := L 0.2,
           M_DO                     := M 2.0);
      NOP   0;
NETWORK
TITLE =
      A     M 2.0;
      =     Q 2.0;
NETWORK
TITLE = осциляція каландр
      A     M 1502.2;
      =     L 0.0;
      BLD   103;
      A     M 1512.2;
      =     L 0.1;
      BLD   103;
      A     M 1522.2;
      =     L 0.2;
      BLD   103;
      CALL  "DO_MANUAL" (
           MANUAL                   := L 0.0,
           PUSK                     := L 0.1,
           STOP                     := L 0.2,
           M_DO                     := M 2.2);
      NOP   0;
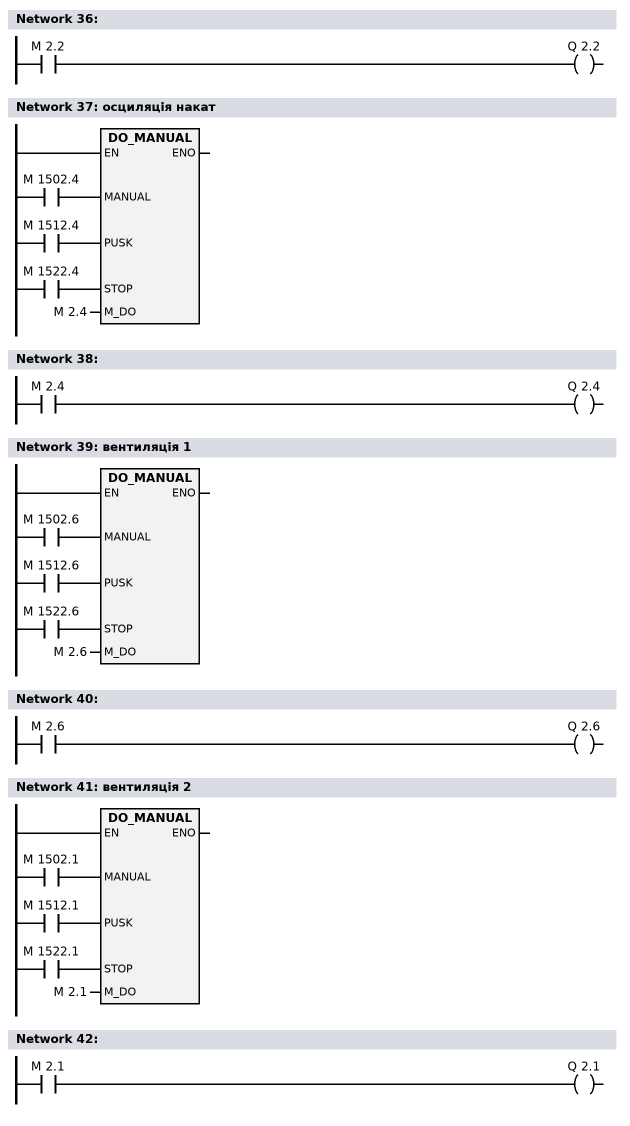
NETWORK
TITLE =
      A     M 2.2;
      =     Q 2.2;
NETWORK
TITLE = осциляція накат
      A     M 1502.4;
      =     L 0.0;
      BLD   103;
      A     M 1512.4;
      =     L 0.1;
      BLD   103;
      A     M 1522.4;
      =     L 0.2;
      BLD   103;
      CALL  "DO_MANUAL" (
           MANUAL                   := L 0.0,
           PUSK                     := L 0.1,
           STOP                     := L 0.2,
           M_DO                     := M 2.4);
      NOP   0;
NETWORK
TITLE =
      A     M 2.4;
      =     Q 2.4;
NETWORK
TITLE = вентиляція 1
      A     M 1502.6;
      =     L 0.0;
      BLD   103;
      A     M 1512.6;
      =     L 0.1;
      BLD   103;
      A     M 1522.6;
      =     L 0.2;
      BLD   103;
      CALL  "DO_MANUAL" (
           MANUAL                   := L 0.0,
           PUSK                     := L 0.1,
           STOP                     := L 0.2,
           M_DO                     := M 2.6);
      NOP   0;
NETWORK
TITLE =
      A     M 2.6;
      =     Q 2.6;
NETWORK
TITLE = вентиляція 2
      A     M 1502.1;
      =     L 0.0;
      BLD   103;
      A     M 1512.1;
      =     L 0.1;
      BLD   103;
      A     M 1522.1;
      =     L 0.2;
      BLD   103;
      CALL  "DO_MANUAL" (
           MANUAL                   := L 0.0,
           PUSK                     := L 0.1,
           STOP                     := L 0.2,
           M_DO                     := M 2.1);
      NOP   0;
NETWORK
TITLE =
      A     M 2.1;
      =     Q 2.1;
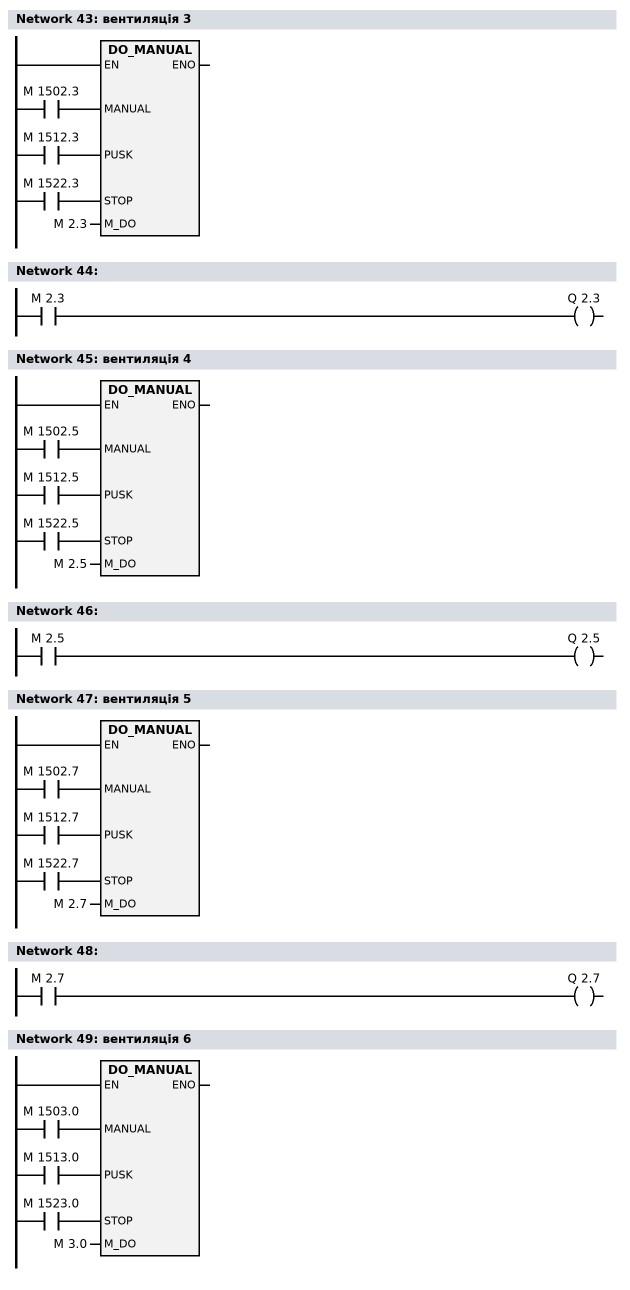
NETWORK
TITLE = вентиляція 3
      A     M 1502.3;
      =     L 0.0;
      BLD   103;
      A     M 1512.3;
      =     L 0.1;
      BLD   103;
      A     M 1522.3;
      =     L 0.2;
      BLD   103;
      CALL  "DO_MANUAL" (
           MANUAL                   := L 0.0,
           PUSK                     := L 0.1,
           STOP                     := L 0.2,
           M_DO                     := M 2.3);
      NOP   0;
NETWORK
TITLE =
      A     M 2.3;
      =     Q 2.3;
NETWORK
TITLE = вентиляція 4
      A     M 1502.5;
      =     L 0.0;
      BLD   103;
      A     M 1512.5;
      =     L 0.1;
      BLD   103;
      A     M 1522.5;
      =     L 0.2;
      BLD   103;
      CALL  "DO_MANUAL" (
           MANUAL                   := L 0.0,
           PUSK                     := L 0.1,
           STOP                     := L 0.2,
           M_DO                     := M 2.5);
      NOP   0;
NETWORK
TITLE =
      A     M 2.5;
      =     Q 2.5;
NETWORK
TITLE = вентиляція 5
      A     M 1502.7;
      =     L 0.0;
      BLD   103;
      A     M 1512.7;
      =     L 0.1;
      BLD   103;
      A     M 1522.7;
      =     L 0.2;
      BLD   103;
      CALL  "DO_MANUAL" (
           MANUAL                   := L 0.0,
           PUSK                     := L 0.1,
           STOP                     := L 0.2,
           M_DO                     := M 2.7);
      NOP   0;
NETWORK
TITLE =
      A     M 2.7;
      =     Q 2.7;
NETWORK
TITLE = вентиляція 6
      A     M 1503.0;
      =     L 0.0;
      BLD   103;
      A     M 1513.0;
      =     L 0.1;
      BLD   103;
      A     M 1523.0;
      =     L 0.2;
      BLD   103;
      CALL  "DO_MANUAL" (
           MANUAL                   := L 0.0,
           PUSK                     := L 0.1,
           STOP                     := L 0.2,
           M_DO                     := M 3.0);
      NOP   0;
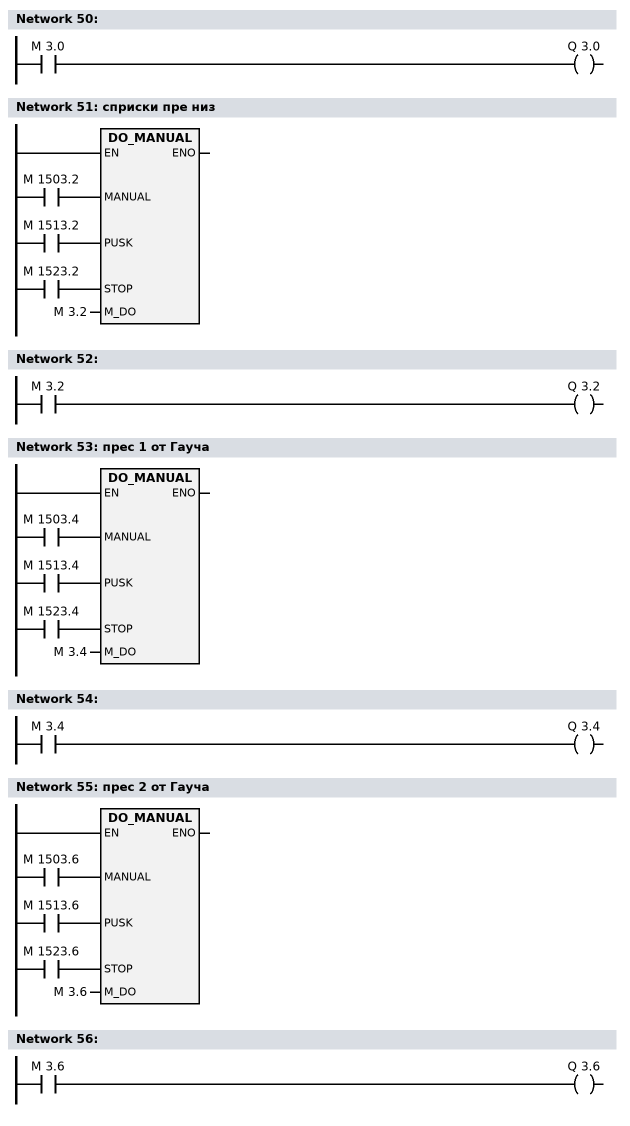
NETWORK
TITLE =
      A     M 3.0;
      =     Q 3.0;
NETWORK
TITLE = сприски пре низ
      A     M 1503.2;
      =     L 0.0;
      BLD   103;
      A     M 1513.2;
      =     L 0.1;
      BLD   103;
      A     M 1523.2;
      =     L 0.2;
      BLD   103;
      CALL  "DO_MANUAL" (
           MANUAL                   := L 0.0,
           PUSK                     := L 0.1,
           STOP                     := L 0.2,
           M_DO                     := M 3.2);
      NOP   0;
NETWORK
TITLE =
      A     M 3.2;
      =     Q 3.2;
NETWORK
TITLE = прес 1 от Гауча
      A     M 1503.4;
      =     L 0.0;
      BLD   103;
      A     M 1513.4;
      =     L 0.1;
      BLD   103;
      A     M 1523.4;
      =     L 0.2;
      BLD   103;
      CALL  "DO_MANUAL" (
           MANUAL                   := L 0.0,
           PUSK                     := L 0.1,
           STOP                     := L 0.2,
           M_DO                     := M 3.4);
      NOP   0;
NETWORK
TITLE =
      A     M 3.4;
      =     Q 3.4;
NETWORK
TITLE = прес 2 от Гауча
      A     M 1503.6;
      =     L 0.0;
      BLD   103;
      A     M 1513.6;
      =     L 0.1;
      BLD   103;
      A     M 1523.6;
      =     L 0.2;
      BLD   103;
      CALL  "DO_MANUAL" (
           MANUAL                   := L 0.0,
           PUSK                     := L 0.1,
           STOP                     := L 0.2,
           M_DO                     := M 3.6);
      NOP   0;
NETWORK
TITLE =
      A     M 3.6;
      =     Q 3.6;
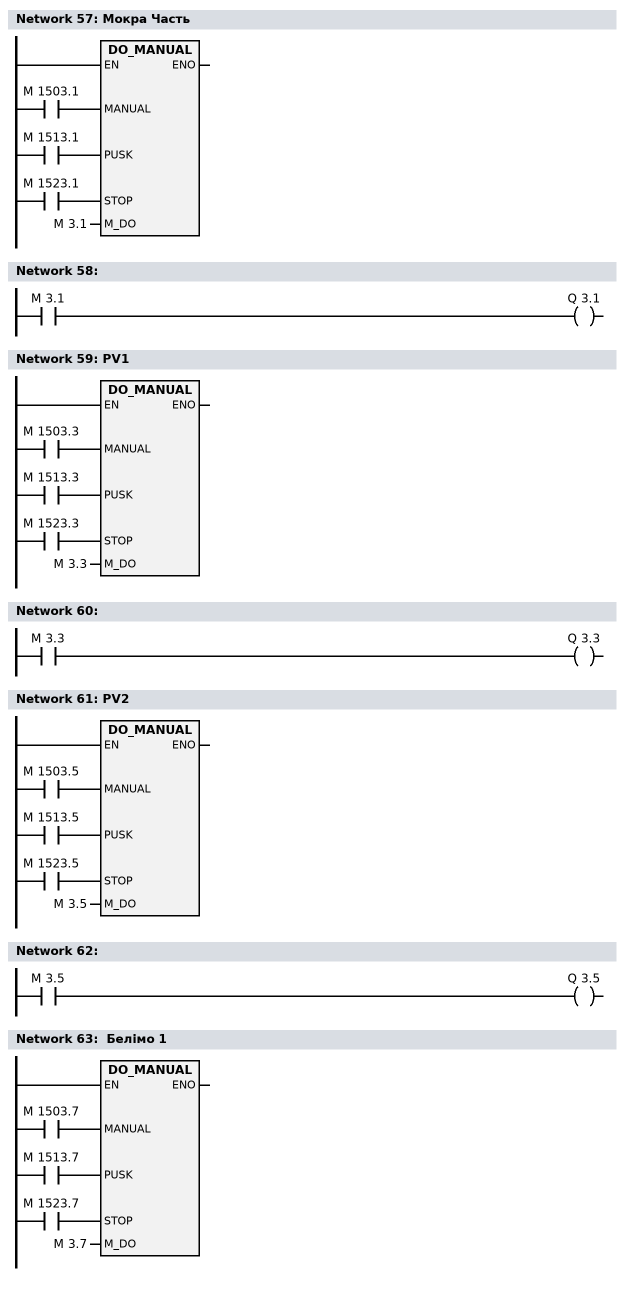
NETWORK
TITLE = Мокра Часть
      A     M 1503.1;
      =     L 0.0;
      BLD   103;
      A     M 1513.1;
      =     L 0.1;
      BLD   103;
      A     M 1523.1;
      =     L 0.2;
      BLD   103;
      CALL  "DO_MANUAL" (
           MANUAL                   := L 0.0,
           PUSK                     := L 0.1,
           STOP                     := L 0.2,
           M_DO                     := M 3.1);
      NOP   0;
NETWORK
TITLE =
      A     M 3.1;
      =     Q 3.1;
NETWORK
TITLE = PV1
      A     M 1503.3;
      =     L 0.0;
      BLD   103;
      A     M 1513.3;
      =     L 0.1;
      BLD   103;
      A     M 1523.3;
      =     L 0.2;
      BLD   103;
      CALL  "DO_MANUAL" (
           MANUAL                   := L 0.0,
           PUSK                     := L 0.1,
           STOP                     := L 0.2,
           M_DO                     := M 3.3);
      NOP   0;
NETWORK
TITLE =
      A     M 3.3;
      =     Q 3.3;
NETWORK
TITLE = PV2
      A     M 1503.5;
      =     L 0.0;
      BLD   103;
      A     M 1513.5;
      =     L 0.1;
      BLD   103;
      A     M 1523.5;
      =     L 0.2;
      BLD   103;
      CALL  "DO_MANUAL" (
           MANUAL                   := L 0.0,
           PUSK                     := L 0.1,
           STOP                     := L 0.2,
           M_DO                     := M 3.5);
      NOP   0;
NETWORK
TITLE =
      A     M 3.5;
      =     Q 3.5;
NETWORK
TITLE =  Белімо 1
      A     M 1503.7;
      =     L 0.0;
      BLD   103;
      A     M 1513.7;
      =     L 0.1;
      BLD   103;
      A     M 1523.7;
      =     L 0.2;
      BLD   103;
      CALL  "DO_MANUAL" (
           MANUAL                   := L 0.0,
           PUSK                     := L 0.1,
           STOP                     := L 0.2,
           M_DO                     := M 3.7);
      NOP   0;
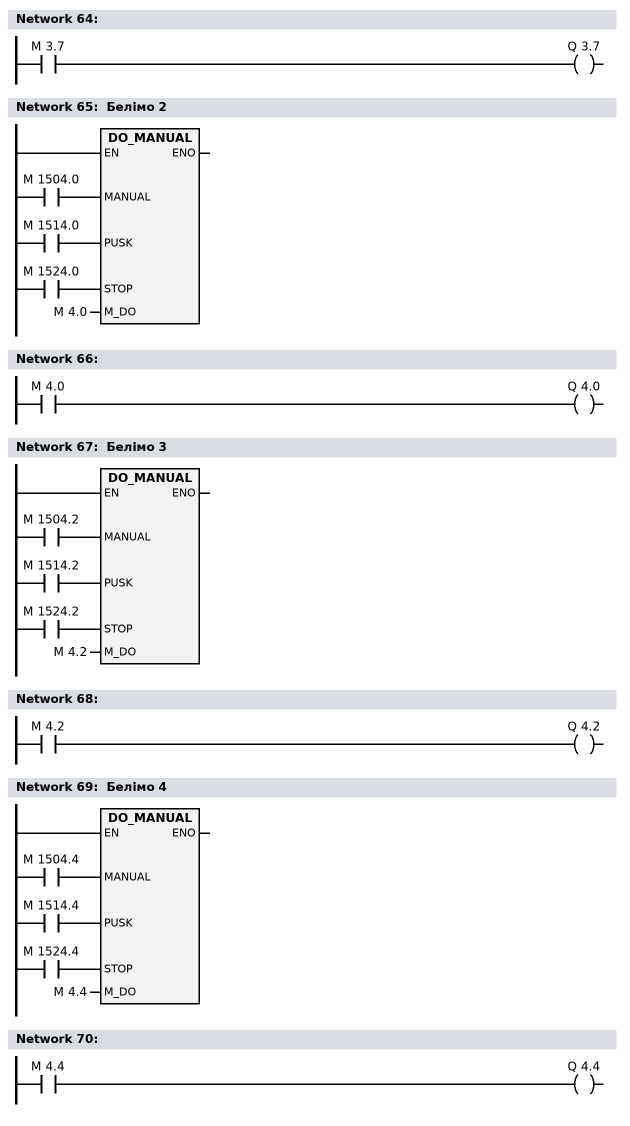
NETWORK
TITLE =
      A     M 3.7;
      =     Q 3.7;
NETWORK
TITLE =  Белімо 2
      A     M 1504.0;
      =     L 0.0;
      BLD   103;
      A     M 1514.0;
      =     L 0.1;
      BLD   103;
      A     M 1524.0;
      =     L 0.2;
      BLD   103;
      CALL  "DO_MANUAL" (
           MANUAL                   := L 0.0,
           PUSK                     := L 0.1,
           STOP                     := L 0.2,
           M_DO                     := M 4.0);
      NOP   0;
NETWORK
TITLE =
      A     M 4.0;
      =     Q 4.0;
NETWORK
TITLE =  Белімо 3
      A     M 1504.2;
      =     L 0.0;
      BLD   103;
      A     M 1514.2;
      =     L 0.1;
      BLD   103;
      A     M 1524.2;
      =     L 0.2;
      BLD   103;
      CALL  "DO_MANUAL" (
           MANUAL                   := L 0.0,
           PUSK                     := L 0.1,
           STOP                     := L 0.2,
           M_DO                     := M 4.2);
      NOP   0;
NETWORK
TITLE =
      A     M 4.2;
      =     Q 4.2;
NETWORK
TITLE =  Белімо 4
      A     M 1504.4;
      =     L 0.0;
      BLD   103;
      A     M 1514.4;
      =     L 0.1;
      BLD   103;
      A     M 1524.4;
      =     L 0.2;
      BLD   103;
      CALL  "DO_MANUAL" (
           MANUAL                   := L 0.0,
           PUSK                     := L 0.1,
           STOP                     := L 0.2,
           M_DO                     := M 4.4);
      NOP   0;
NETWORK
TITLE =
      A     M 4.4;
      =     Q 4.4;
END_FUNCTION_BLOCK

FUNCTION_BLOCK "DI_DO_STATE"	// FB 4
//DI DO State for NetSend
VERSION : 0.1
BEGIN
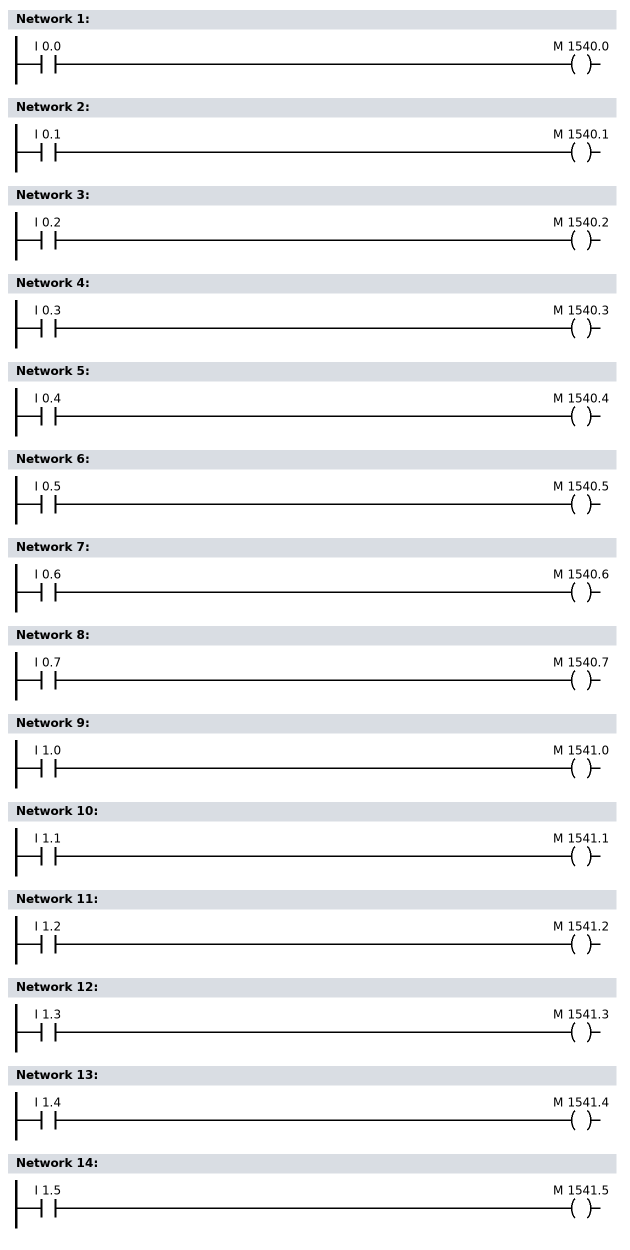
NETWORK
TITLE =
//Стан входів для обміну по мережі
      A     I 0.0;
      =     M 1540.0;
NETWORK
TITLE =
      A     I 0.1;
      =     M 1540.1;
NETWORK
TITLE =
      A     I 0.2;
      =     M 1540.2;
NETWORK
TITLE =
      A     I 0.3;
      =     M 1540.3;
NETWORK
TITLE =
      A     I 0.4;
      =     M 1540.4;
NETWORK
TITLE =
      A     I 0.5;
      =     M 1540.5;
NETWORK
TITLE =
      A     I 0.6;
      =     M 1540.6;
NETWORK
TITLE =
      A     I 0.7;
      =     M 1540.7;
NETWORK
TITLE =
      A     I 1.0;
      =     M 1541.0;
NETWORK
TITLE =
      A     I 1.1;
      =     M 1541.1;
NETWORK
TITLE =
      A     I 1.2;
      =     M 1541.2;
NETWORK
TITLE =
      A     I 1.3;
      =     M 1541.3;
NETWORK
TITLE =
      A     I 1.4;
      =     M 1541.4;
NETWORK
TITLE =
      A     I 1.5;
      =     M 1541.5;
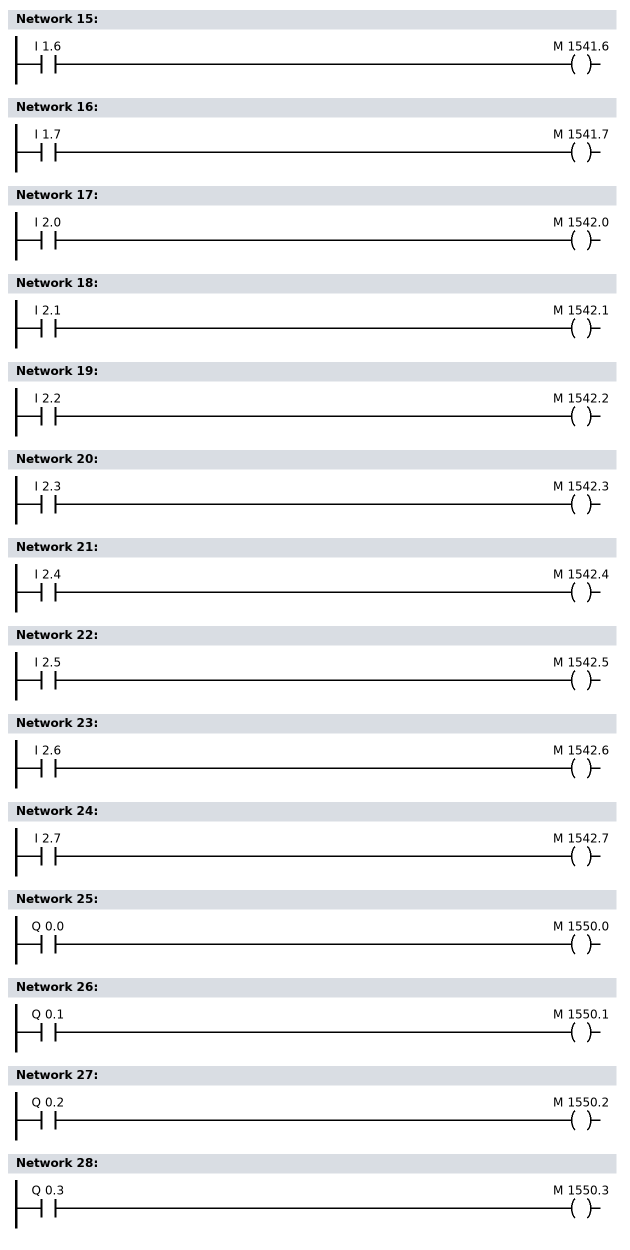
NETWORK
TITLE =
      A     I 1.6;
      =     M 1541.6;
NETWORK
TITLE =
      A     I 1.7;
      =     M 1541.7;
NETWORK
TITLE =
      A     I 2.0;
      =     M 1542.0;
NETWORK
TITLE =
      A     I 2.1;
      =     M 1542.1;
NETWORK
TITLE =
      A     I 2.2;
      =     M 1542.2;
NETWORK
TITLE =
      A     I 2.3;
      =     M 1542.3;
NETWORK
TITLE =
      A     I 2.4;
      =     M 1542.4;
NETWORK
TITLE =
      A     I 2.5;
      =     M 1542.5;
NETWORK
TITLE =
      A     I 2.6;
      =     M 1542.6;
NETWORK
TITLE =
      A     I 2.7;
      =     M 1542.7;
NETWORK
TITLE =
//Стан виходів для обміну по мережі
      A     Q 0.0;
      =     M 1550.0;
NETWORK
TITLE =
      A     Q 0.1;
      =     M 1550.1;
NETWORK
TITLE =
      A     Q 0.2;
      =     M 1550.2;
NETWORK
TITLE =
      A     Q 0.3;
      =     M 1550.3;
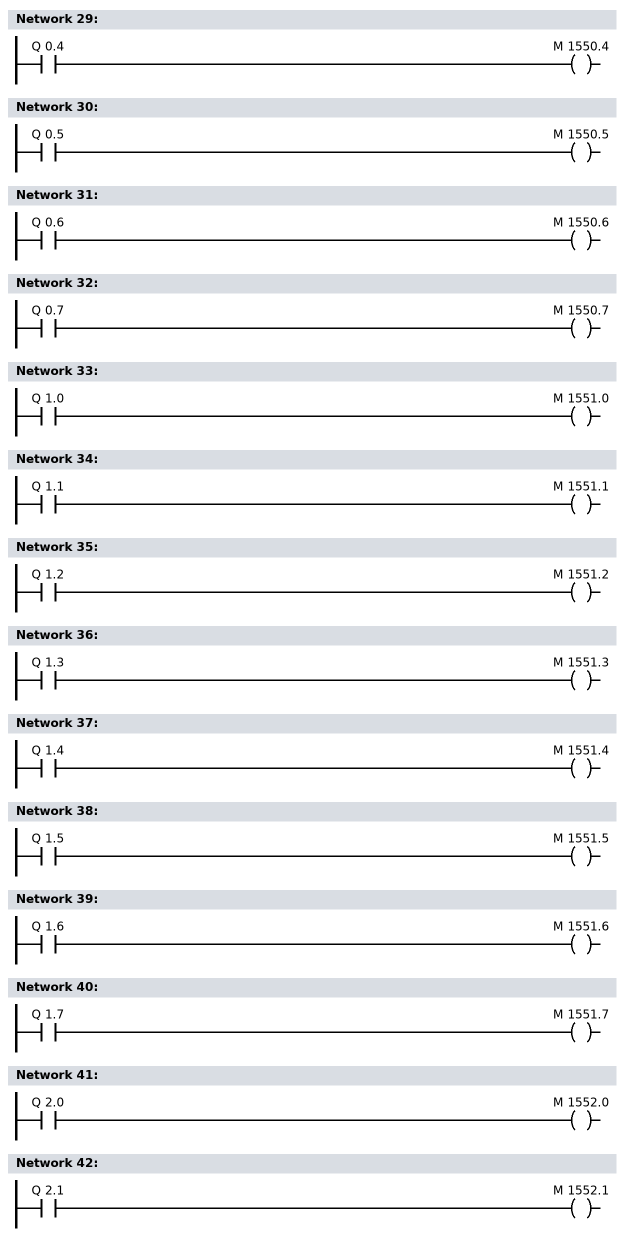
NETWORK
TITLE =
      A     Q 0.4;
      =     M 1550.4;
NETWORK
TITLE =
      A     Q 0.5;
      =     M 1550.5;
NETWORK
TITLE =
      A     Q 0.6;
      =     M 1550.6;
NETWORK
TITLE =
      A     Q 0.7;
      =     M 1550.7;
NETWORK
TITLE =
      A     Q 1.0;
      =     M 1551.0;
NETWORK
TITLE =
      A     Q 1.1;
      =     M 1551.1;
NETWORK
TITLE =
      A     Q 1.2;
      =     M 1551.2;
NETWORK
TITLE =
      A     Q 1.3;
      =     M 1551.3;
NETWORK
TITLE =
      A     Q 1.4;
      =     M 1551.4;
NETWORK
TITLE =
      A     Q 1.5;
      =     M 1551.5;
NETWORK
TITLE =
      A     Q 1.6;
      =     M 1551.6;
NETWORK
TITLE =
      A     Q 1.7;
      =     M 1551.7;
NETWORK
TITLE =
      A     Q 2.0;
      =     M 1552.0;
NETWORK
TITLE =
      A     Q 2.1;
      =     M 1552.1;
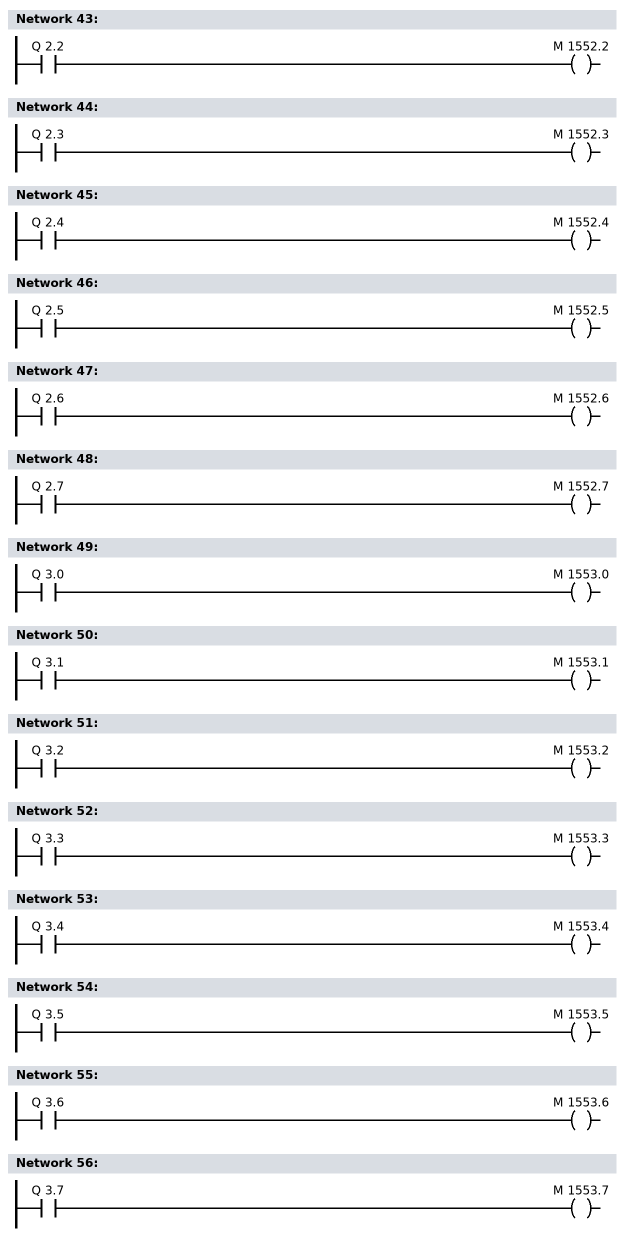
NETWORK
TITLE =
      A     Q 2.2;
      =     M 1552.2;
NETWORK
TITLE =
      A     Q 2.3;
      =     M 1552.3;
NETWORK
TITLE =
      A     Q 2.4;
      =     M 1552.4;
NETWORK
TITLE =
      A     Q 2.5;
      =     M 1552.5;
NETWORK
TITLE =
      A     Q 2.6;
      =     M 1552.6;
NETWORK
TITLE =
      A     Q 2.7;
      =     M 1552.7;
NETWORK
TITLE =
      A     Q 3.0;
      =     M 1553.0;
NETWORK
TITLE =
      A     Q 3.1;
      =     M 1553.1;
NETWORK
TITLE =
      A     Q 3.2;
      =     M 1553.2;
NETWORK
TITLE =
      A     Q 3.3;
      =     M 1553.3;
NETWORK
TITLE =
      A     Q 3.4;
      =     M 1553.4;
NETWORK
TITLE =
      A     Q 3.5;
      =     M 1553.5;
NETWORK
TITLE =
      A     Q 3.6;
      =     M 1553.6;
NETWORK
TITLE =
      A     Q 3.7;
      =     M 1553.7;
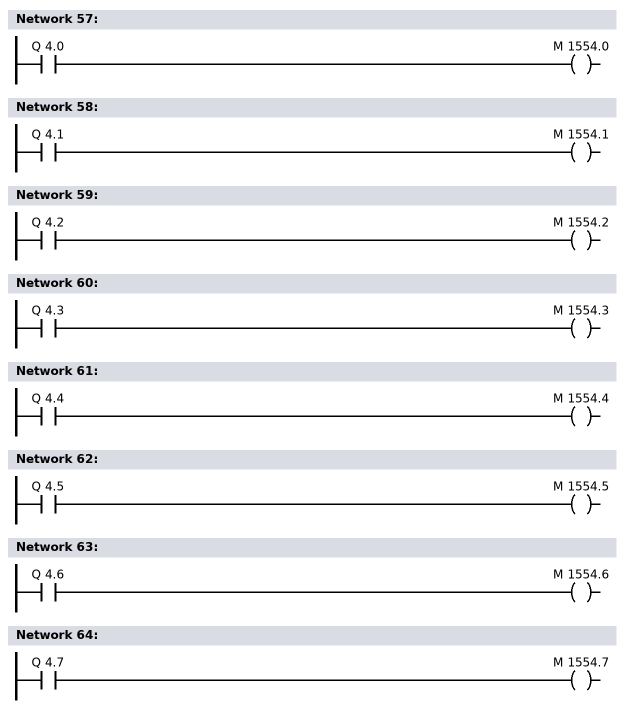
NETWORK
TITLE =
      A     Q 4.0;
      =     M 1554.0;
NETWORK
TITLE =
      A     Q 4.1;
      =     M 1554.1;
NETWORK
TITLE =
      A     Q 4.2;
      =     M 1554.2;
NETWORK
TITLE =
      A     Q 4.3;
      =     M 1554.3;
NETWORK
TITLE =
      A     Q 4.4;
      =     M 1554.4;
NETWORK
TITLE =
      A     Q 4.5;
      =     M 1554.5;
NETWORK
TITLE =
      A     Q 4.6;
      =     M 1554.6;
NETWORK
TITLE =
      A     Q 4.7;
      =     M 1554.7;
END_FUNCTION_BLOCK

FUNCTION_BLOCK "PID_AO_control"	// FB 5
TITLE = параметры PID + управление аналоговым выходом (AO)
//параметры PID + управление аналоговым выходом (AO)
VERSION : 0.1
VAR_INPUT
  Dat_err : BOOL ;
  Dat_re : REAL ;
  P_dw : DWORD ;
  I_dw : DWORD ;
  D_dw : DWORD ;
  TASK_dw : DWORD ;
  PID_LMN : REAL ;
END_VAR
VAR_OUTPUT
  TASK_pid : REAL ;
  PV_pid : REAL ;
  P_pid : REAL ;
  I_pid : REAL ;
  D_pid : REAL ;
  AO_PQW : INT ;
  AO_md : DWORD ;
END_VAR
VAR
  Bipolar : BOOL ;
  AO_val : INT ;
END_VAR
VAR_TEMP
  UNSCL_err : WORD ;
END_VAR
BEGIN
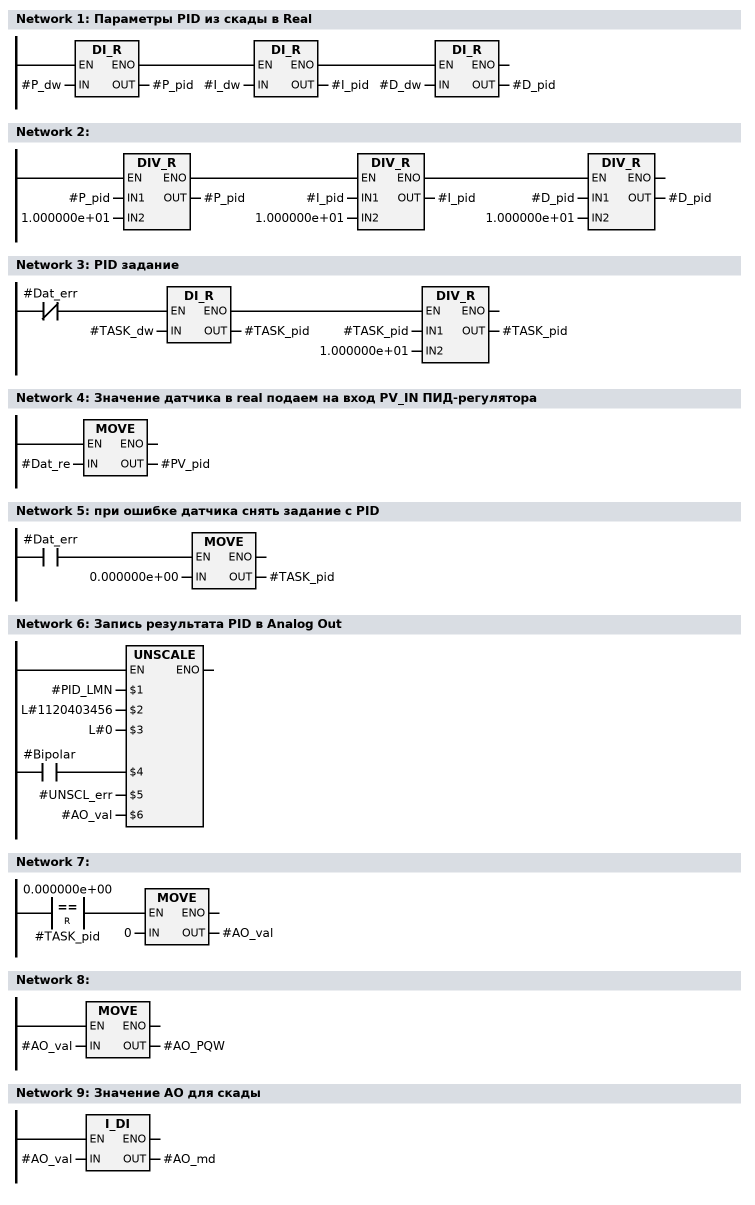
NETWORK
TITLE = Параметры PID из скады в Real
//********************************************************************************
//
      A(;
      A(;
      L     #P_dw;
      DTR;
      T     #P_pid;
      SET;
      SAVE;
      CLR;
      A     BR;
      );
      JNB   _001;
      L     #I_dw;
      DTR;
      T     #I_pid;
      SET;
      SAVE;
      CLR;
_001: A     BR;
      );
      JNB   _002;
      L     #D_dw;
      DTR;
      T     #D_pid;
_002: NOP   0;
NETWORK
TITLE =
      A(;
      A(;
      L     #P_pid;
      L     1.000000e+01;
      /R;
      T     #P_pid;
      AN    OV;
      SAVE;
      CLR;
      A     BR;
      );
      JNB   _007;
      L     #I_pid;
      L     1.000000e+01;
      /R;
      T     #I_pid;
      AN    OV;
      SAVE;
      CLR;
_007: A     BR;
      );
      JNB   _008;
      L     #D_pid;
      L     1.000000e+01;
      /R;
      T     #D_pid;
_008: NOP   0;
NETWORK
TITLE = PID задание
      A(;
      AN    #Dat_err;
      JNB   _009;
      L     #TASK_dw;
      DTR;
      T     #TASK_pid;
      SET;
      SAVE;
      CLR;
_009: A     BR;
      );
      JNB   _00a;
      L     #TASK_pid;
      L     1.000000e+01;
      /R;
      T     #TASK_pid;
_00a: NOP   0;
NETWORK
TITLE = Значение датчика в real подаем на вход PV_IN ПИД-регулятора
      L     #Dat_re;
      T     #PV_pid;
      NOP   0;
NETWORK
TITLE = при ошибке датчика снять задание с PID
      A     #Dat_err;
      JNB   _00b;
      L     0.000000e+00;
      T     #TASK_pid;
_00b: NOP   0;
NETWORK
TITLE = Запись результата PID в Analog Out
      A     #Bipolar;
      =     L 2.0;
      BLD   103;
      CALL  "UNSCALE" (
           $1                       := #PID_LMN,
           $2                       := L#1120403456,
           $3                       := L#0,
           $4                       := L 2.0,
           $5                       := #UNSCL_err,
           $6                       := #AO_val);
      NOP   0;
NETWORK
TITLE =
//Если задание 0, то записать 0 в значение AO
//
      A(;
      L     0.000000e+00;
      L     #TASK_pid;
      ==R;
      );
      JNB   _00c;
      L     0;
      T     #AO_val;
_00c: NOP   0;
NETWORK
TITLE =
      L     #AO_val;
      T     #AO_PQW;
      NOP   0;
NETWORK
TITLE = Значение AO для скады
      L     #AO_val;
      ITD;
      T     #AO_md;
      NOP   0;
END_FUNCTION_BLOCK

FUNCTION_BLOCK "dat_alm"	// FB 6
TITLE = Dat_Alarm
//Аварія max, Попередження max, Попередження min, Аварія min
VERSION : 0.1
BEGIN
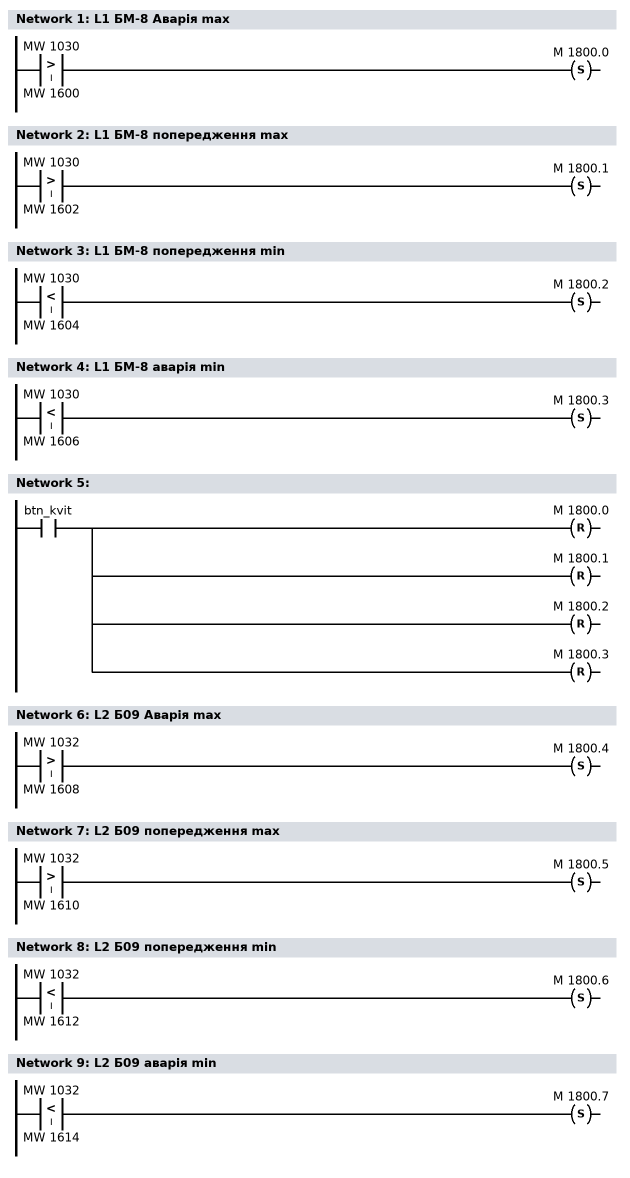
NETWORK
TITLE = L1 БМ-8 Аварія max
      L     MW 1030;
      L     MW 1600;
      >I;
      S     M 1800.0;
NETWORK
TITLE = L1 БМ-8 попередження max
      L     MW 1030;
      L     MW 1602;
      >I;
      S     M 1800.1;
NETWORK
TITLE = L1 БМ-8 попередження min
      L     MW 1030;
      L     MW 1604;
      <I;
      S     M 1800.2;
NETWORK
TITLE = L1 БМ-8 аварія min
      L     MW 1030;
      L     MW 1606;
      <I;
      S     M 1800.3;
NETWORK
TITLE =
      A     "btn_kvit";
      R     M 1800.0;
      R     M 1800.1;
      R     M 1800.2;
      R     M 1800.3;
NETWORK
TITLE = L2 Б09 Аварія max
//*************************************************
      L     MW 1032;
      L     MW 1608;
      >I;
      S     M 1800.4;
NETWORK
TITLE = L2 Б09 попередження max
      L     MW 1032;
      L     MW 1610;
      >I;
      S     M 1800.5;
NETWORK
TITLE = L2 Б09 попередження min
      L     MW 1032;
      L     MW 1612;
      <I;
      S     M 1800.6;
NETWORK
TITLE = L2 Б09 аварія min
      L     MW 1032;
      L     MW 1614;
      <I;
      S     M 1800.7;
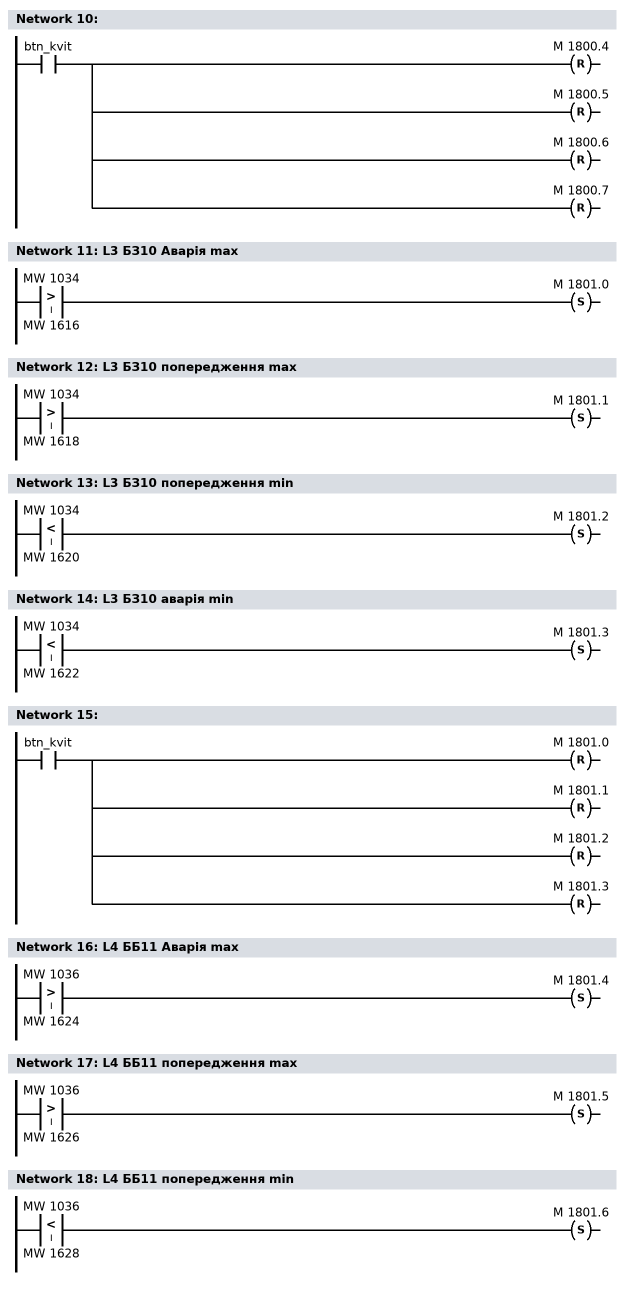
NETWORK
TITLE =
      A     "btn_kvit";
      R     M 1800.4;
      R     M 1800.5;
      R     M 1800.6;
      R     M 1800.7;
NETWORK
TITLE = L3 БЗ10 Аварія max
//*************************************************
      L     MW 1034;
      L     MW 1616;
      >I;
      S     M 1801.0;
NETWORK
TITLE = L3 БЗ10 попередження max
      L     MW 1034;
      L     MW 1618;
      >I;
      S     M 1801.1;
NETWORK
TITLE = L3 БЗ10 попередження min
      L     MW 1034;
      L     MW 1620;
      <I;
      S     M 1801.2;
NETWORK
TITLE = L3 БЗ10 аварія min
      L     MW 1034;
      L     MW 1622;
      <I;
      S     M 1801.3;
NETWORK
TITLE =
      A     "btn_kvit";
      R     M 1801.0;
      R     M 1801.1;
      R     M 1801.2;
      R     M 1801.3;
NETWORK
TITLE = L4 ББ11 Аварія max
//*************************************************
      L     MW 1036;
      L     MW 1624;
      >I;
      S     M 1801.4;
NETWORK
TITLE = L4 ББ11 попередження max
      L     MW 1036;
      L     MW 1626;
      >I;
      S     M 1801.5;
NETWORK
TITLE = L4 ББ11 попередження min
      L     MW 1036;
      L     MW 1628;
      <I;
      S     M 1801.6;
